KUKA KRL program: MyProgram_010().src

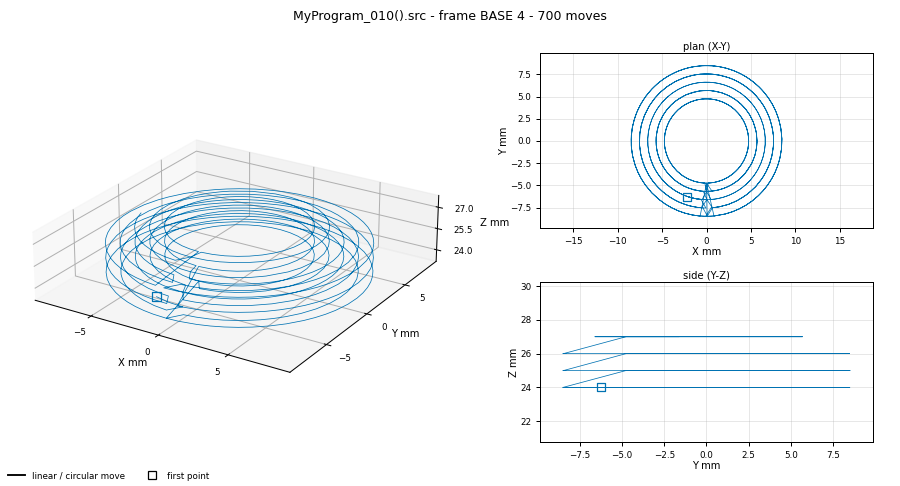
[picture p0: tool path of MyProgram_010().src in frame BASE 4, 700 of 700 moves have a stored position in this frame; points joined in program order, loops and branches not executed]
&ACCESS RVP
&REL 1
&PARAM TEMPLATE = C:\KRC\Roboter\Template\vorgabe
&PARAM EDITMASK = *
DEF MyProgram_010()
; ---- Setting reference (Base) ----
$BASE = BASE_DATA[4]

; --------------------------
; ---- Setting tool (TCP) ----
$TOOL = TOOL_DATA[3]
; --------------------------

$VEL.CP = VEL_APROX_PRINT
Startdeposition()
$VEL.CP = VEL_PRINT
LIN {X -2.1509,Y -6.2604,Z 24,A -3.0859,B 0,C 0,E1 0.1598,E2 90.0714} C_DIS
LIN {X -1.1022,Y -6.531,Z 24,A -3.0589,B 0,C 0,E1 0.1598,E2 90.0714} C_DIS
LIN {X 0.0303,Y -6.6205,Z 24,A -3.0212,B 0,C 0,E1 0.1598,E2 90.0715} C_DIS
Enddeposition()
LIN {X 0.0303,Y -6.6205,Z 24,A -3.0212,B 0,C 0,E1 0.1598,E2 90.0715} C_DIS
Startdeposition()
$VEL.CP = VEL_PRINT
LIN {X -0.5711,Y -7.5301,Z 24,A -3.0815,B 0,C 0,E1 0.1598,E2 90.0709} C_DIS
LIN {X -1.5725,Y -7.3914,Z 24,A -3.1128,B 0,C 0,E1 0.1598,E2 90.0714} C_DIS
LIN {X -2.6511,Y -7.0725,Z 24,A -3.1389,B 0,C 0,E1 0.1598,E2 90.0714} C_DIS
LIN {X -3.396,Y -6.7456,Z 24,A -3.1523,B 0,C 0,E1 0.1598,E2 90.0714} C_DIS
LIN {X -4.1021,Y -6.3418,Z 24,A -3.1611,B 0,C 0,E1 0.1598,E2 90.0713} C_DIS
LIN {X -4.7604,Y -5.8639,Z 24,A -3.165,B 0,C 0,E1 0.1598,E2 90.0713} C_DIS
LIN {X -5.3635,Y -5.318,Z 24,A -3.164,B 0,C 0,E1 0.1598,E2 90.0712} C_DIS
LIN {X -5.9042,Y -4.7103,Z 24,A -3.1581,B 0,C 0,E1 0.1598,E2 90.0712} C_DIS
LIN {X -6.3764,Y -4.048,Z 24,A -3.1474,B 0,C 0,E1 0.1598,E2 90.0712} C_DIS
LIN {X -6.7752,Y -3.339,Z 24,A -3.1321,B 0,C 0,E1 0.1598,E2 90.0712} C_DIS
LIN {X -7.1999,Y -2.2947,Z 24,A -3.1033,B 0,C 0,E1 0.1598,E2 90.0709} C_DIS
LIN {X -7.4401,Y -1.3287,Z 24,A -3.0713,B 0,C 0,E1 0.1598,E2 90.0709} C_DIS
LIN {X -7.5468,Y -0.4046,Z 24,A -3.0364,B 0,C 0,E1 0.1598,E2 90.0711} C_DIS
LIN {X -7.5022,Y 0.9089,Z 24,A -2.9788,B 0,C 0,E1 0.1598,E2 90.0706} C_DIS
LIN {X -7.3211,Y 1.8726,Z 24,A -2.9319,B 0,C 0,E1 0.1598,E2 90.0711} C_DIS
LIN {X -6.9098,Y 3.0609,Z 24,A -2.8664,B 0,C 0,E1 0.1598,E2 90.0711} C_DIS
LIN {X -6.4301,Y 3.9691,Z 24,A -2.8107,B 0,C 0,E1 0.1598,E2 90.0714} C_DIS
LIN {X -5.7251,Y 4.9319,Z 24,A -2.7441,B 0,C 0,E1 0.1598,E2 90.0714} C_DIS
LIN {X -5.1328,Y 5.5464,Z 24,A -2.6965,B 0,C 0,E1 0.1598,E2 90.0717} C_DIS
LIN {X -4.2881,Y 6.2219,Z 24,A -2.6369,B 0,C 0,E1 0.1598,E2 90.0718} C_DIS
LIN {X -3.4726,Y 6.7132,Z 24,A -2.5862,B 0,C 0,E1 0.1598,E2 90.072} C_DIS
LIN {X -2.6704,Y 7.0647,Z 24,A -2.5418,B 0,C 0,E1 0.1598,E2 90.0721} C_DIS
LIN {X -1.6242,Y 7.3805,Z 24,A -2.4898,B 0,C 0,E1 0.1598,E2 90.0722} C_DIS
LIN {X -0.7055,Y 7.5252,Z 24,A -2.4498,B 0,C 0,E1 0.1598,E2 90.0722} C_DIS
LIN {X 0.503,Y 7.5401,Z 24,A -2.4046,B 0,C 0,E1 0.1598,E2 90.0724} C_DIS
LIN {X 1.3896,Y 7.4296,Z 24,A -2.3765,B 0,C 0,E1 0.1598,E2 90.0724} C_DIS
LIN {X 2.6317,Y 7.0805,Z 24,A -2.3454,B 0,C 0,E1 0.1598,E2 90.0724} C_DIS
LIN {X 3.395,Y 6.7468,Z 24,A -2.3314,B 0,C 0,E1 0.1598,E2 90.0724} C_DIS
LIN {X 4.1176,Y 6.3321,Z 24,A -2.3223,B 0,C 0,E1 0.1598,E2 90.0724} C_DIS
LIN {X 4.7897,Y 5.8397,Z 24,A -2.3183,B 0,C 0,E1 0.1598,E2 90.0724} C_DIS
LIN {X 5.6394,Y 5.032,Z 24,A -2.321,B 0,C 0,E1 0.1598,E2 90.0721} C_DIS
LIN {X 6.3129,Y 4.149,Z 24,A -2.3336,B 0,C 0,E1 0.1598,E2 90.0721} C_DIS
LIN {X 6.6648,Y 3.5575,Z 24,A -2.346,B 0,C 0,E1 0.1598,E2 90.0722} C_DIS
LIN {X 7.0965,Y 2.5964,Z 24,A -2.3706,B 0,C 0,E1 0.1598,E2 90.0719} C_DIS
LIN {X 7.4222,Y 1.4016,Z 24,A -2.4091,B 0,C 0,E1 0.1598,E2 90.0715} C_DIS
LIN {X 7.5337,Y 0.5498,Z 24,A -2.4417,B 0,C 0,E1 0.1598,E2 90.0719} C_DIS
LIN {X 7.5455,Y -0.3091,Z 24,A -2.4778,B 0,C 0,E1 0.1598,E2 90.0719} C_DIS
LIN {X 7.4322,Y -1.3766,Z 24,A -2.5271,B 0,C 0,E1 0.1598,E2 90.0715} C_DIS
LIN {X 7.1168,Y -2.5308,Z 24,A -2.5877,B 0,C 0,E1 0.1598,E2 90.0713} C_DIS
LIN {X 6.6477,Y -3.5933,Z 24,A -2.6504,B 0,C 0,E1 0.1598,E2 90.0715} C_DIS
LIN {X 6.1054,Y -4.445,Z 24,A -2.7067,B 0,C 0,E1 0.1598,E2 90.0716} C_DIS
LIN {X 5.5965,Y -5.0722,Z 24,A -2.7522,B 0,C 0,E1 0.1598,E2 90.0716} C_DIS
LIN {X 5.0229,Y -5.641,Z 24,A -2.7975,B 0,C 0,E1 0.1598,E2 90.0716} C_DIS
LIN {X 4.1409,Y -6.3233,Z 24,A -2.8589,B 0,C 0,E1 0.1598,E2 90.0716} C_DIS
LIN {X 3.1206,Y -6.8785,Z 24,A -2.92,B 0,C 0,E1 0.1598,E2 90.0716} C_DIS
LIN {X 2.3301,Y -7.1857,Z 24,A -2.9621,B 0,C 0,E1 0.1598,E2 90.0716} C_DIS
LIN {X 1.5095,Y -7.3999,Z 24,A -3.0013,B 0,C 0,E1 0.1598,E2 90.0716} C_DIS
LIN {X 0.6704,Y -7.5218,Z 24,A -3.0373,B 0,C 0,E1 0.1598,E2 90.0716} C_DIS
LIN {X 0.6704,Y -7.5218,Z 24,A -3.0373,B 0,C 0,E1 0.1598,E2 90.0716} C_DIS
Enddeposition()
LIN {X 0.0638,Y -8.4902,Z 24,A -3.0997,B 0,C 0,E1 0.1598,E2 90.0703} C_DIS
Startdeposition()
$VEL.CP = VEL_PRINT
LIN {X 0.9236,Y -8.4401,Z 24,A -3.0671,B 0,C 0,E1 0.1598,E2 90.0714} C_DIS
LIN {X 2.0955,Y -8.2263,Z 24,A -3.0151,B 0,C 0,E1 0.1598,E2 90.0715} C_DIS
LIN {X 2.906,Y -7.9764,Z 24,A -2.9748,B 0,C 0,E1 0.1598,E2 90.0715} C_DIS
LIN {X 3.6874,Y -7.6466,Z 24,A -2.9321,B 0,C 0,E1 0.1598,E2 90.0716} C_DIS
LIN {X 4.432,Y -7.2405,Z 24,A -2.8875,B 0,C 0,E1 0.1598,E2 90.0716} C_DIS
LIN {X 5.1322,Y -6.7618,Z 24,A -2.8414,B 0,C 0,E1 0.1598,E2 90.0716} C_DIS
LIN {X 5.9363,Y -6.0709,Z 24,A -2.7823,B 0,C 0,E1 0.1598,E2 90.0716} C_DIS
LIN {X 6.6411,Y -5.2912,Z 24,A -2.7233,B 0,C 0,E1 0.1598,E2 90.0716} C_DIS
LIN {X 7.2908,Y -4.3455,Z 24,A -2.659,B 0,C 0,E1 0.1598,E2 90.0716} C_DIS
LIN {X 7.6767,Y -3.6219,Z 24,A -2.6142,B 0,C 0,E1 0.1598,E2 90.0718} C_DIS
LIN {X 7.9908,Y -2.8643,Z 24,A -2.5703,B 0,C 0,E1 0.1598,E2 90.0718} C_DIS
LIN {X 8.2302,Y -2.0798,Z 24,A -2.5281,B 0,C 0,E1 0.1598,E2 90.0718} C_DIS
LIN {X 8.4401,Y -0.9236,Z 24,A -2.4708,B 0,C 0,E1 0.1598,E2 90.0716} C_DIS
LIN {X 8.4863,Y 0.148,Z 24,A -2.4236,B 0,C 0,E1 0.1598,E2 90.0717} C_DIS
LIN {X 8.4278,Y 1.004,Z 24,A -2.3894,B 0,C 0,E1 0.1598,E2 90.072} C_DIS
LIN {X 8.2824,Y 1.8497,Z 24,A -2.3588,B 0,C 0,E1 0.1598,E2 90.072} C_DIS
LIN {X 8.0532,Y 2.6767,Z 24,A -2.3321,B 0,C 0,E1 0.1598,E2 90.072} C_DIS
LIN {X 7.7419,Y 3.4763,Z 24,A -2.3096,B 0,C 0,E1 0.1598,E2 90.0721} C_DIS
LIN {X 7.3514,Y 4.2404,Z 24,A -2.2915,B 0,C 0,E1 0.1598,E2 90.0721} C_DIS
LIN {X 6.8858,Y 4.9613,Z 24,A -2.2781,B 0,C 0,E1 0.1598,E2 90.0722} C_DIS
LIN {X 6.2076,Y 5.7923,Z 24,A -2.2676,B 0,C 0,E1 0.1598,E2 90.0721} C_DIS
LIN {X 5.4453,Y 6.5144,Z 24,A -2.2652,B 0,C 0,E1 0.1598,E2 90.0722} C_DIS
LIN {X 4.4548,Y 7.2234,Z 24,A -2.2717,B 0,C 0,E1 0.1598,E2 90.0722} C_DIS
LIN {X 3.733,Y 7.6202,Z 24,A -2.2817,B 0,C 0,E1 0.1598,E2 90.0724} C_DIS
LIN {X 2.9768,Y 7.9466,Z 24,A -2.2959,B 0,C 0,E1 0.1598,E2 90.0724} C_DIS
LIN {X 2.1925,Y 8.1983,Z 24,A -2.3142,B 0,C 0,E1 0.1598,E2 90.0724} C_DIS
LIN {X 1.3875,Y 8.3731,Z 24,A -2.3366,B 0,C 0,E1 0.1598,E2 90.0724} C_DIS
LIN {X 0.5694,Y 8.4695,Z 24,A -2.3627,B 0,C 0,E1 0.1598,E2 90.0724} C_DIS
LIN {X -0.4602,Y 8.4788,Z 24,A -2.4003,B 0,C 0,E1 0.1598,E2 90.0724} C_DIS
LIN {X -1.7187,Y 8.3132,Z 24,A -2.4538,B 0,C 0,E1 0.1598,E2 90.0723} C_DIS
LIN {X -2.5445,Y 8.0987,Z 24,A -2.4933,B 0,C 0,E1 0.1598,E2 90.0723} C_DIS
LIN {X -3.3445,Y 7.8021,Z 24,A -2.5354,B 0,C 0,E1 0.1598,E2 90.0722} C_DIS
LIN {X -4.1107,Y 7.4269,Z 24,A -2.5795,B 0,C 0,E1 0.1598,E2 90.0721} C_DIS
LIN {X -4.8354,Y 6.9766,Z 24,A -2.6252,B 0,C 0,E1 0.1598,E2 90.072} C_DIS
LIN {X -5.5111,Y 6.4557,Z 24,A -2.672,B 0,C 0,E1 0.1598,E2 90.0719} C_DIS
LIN {X -6.1312,Y 5.8697,Z 24,A -2.7196,B 0,C 0,E1 0.1598,E2 90.0718} C_DIS
LIN {X -6.8215,Y 5.0568,Z 24,A -2.7791,B 0,C 0,E1 0.1598,E2 90.0715} C_DIS
LIN {X -7.3978,Y 4.1667,Z 24,A -2.8378,B 0,C 0,E1 0.1598,E2 90.0714} C_DIS
LIN {X -7.8737,Y 3.1665,Z 24,A -2.8975,B 0,C 0,E1 0.1598,E2 90.0713} C_DIS
LIN {X -8.1612,Y 2.3284,Z 24,A -2.9435,B 0,C 0,E1 0.1598,E2 90.0713} C_DIS
LIN {X -8.3602,Y 1.4649,Z 24,A -2.9872,B 0,C 0,E1 0.1598,E2 90.0713} C_DIS
LIN {X -8.4687,Y 0.5855,Z 24,A -3.0282,B 0,C 0,E1 0.1598,E2 90.0711} C_DIS
LIN {X -8.4746,Y -0.5221,Z 24,A -3.0748,B 0,C 0,E1 0.1598,E2 90.0707} C_DIS
LIN {X -8.343,Y -1.5835,Z 24,A -3.1148,B 0,C 0,E1 0.1598,E2 90.0708} C_DIS
LIN {X -8.0507,Y -2.6866,Z 24,A -3.1506,B 0,C 0,E1 0.1598,E2 90.0707} C_DIS
LIN {X -7.7407,Y -3.4806,Z 24,A -3.173,B 0,C 0,E1 0.1598,E2 90.071} C_DIS
LIN {X -7.3527,Y -4.2396,Z 24,A -3.1909,B 0,C 0,E1 0.1598,E2 90.071} C_DIS
LIN {X -6.8904,Y -4.9557,Z 24,A -3.2042,B 0,C 0,E1 0.1598,E2 90.071} C_DIS
LIN {X -6.2176,Y -5.7818,Z 24,A -3.2143,B 0,C 0,E1 0.1598,E2 90.0709} C_DIS
LIN {X -5.4465,Y -6.5135,Z 24,A -3.217,B 0,C 0,E1 0.1598,E2 90.0709} C_DIS
LIN {X -4.6444,Y -7.103,Z 24,A -3.2127,B 0,C 0,E1 0.1598,E2 90.0711} C_DIS
LIN {X -3.9579,Y -7.5063,Z 24,A -3.2047,B 0,C 0,E1 0.1598,E2 90.0712} C_DIS
LIN {X -3.2368,Y -7.8438,Z 24,A -3.1926,B 0,C 0,E1 0.1598,E2 90.0712} C_DIS
LIN {X -2.4874,Y -8.1126,Z 24,A -3.1765,B 0,C 0,E1 0.1598,E2 90.0712} C_DIS
LIN {X -1.7162,Y -8.3104,Z 24,A -3.1567,B 0,C 0,E1 0.1598,E2 90.0713} C_DIS
LIN {X -0.9299,Y -8.4356,Z 24,A -3.1332,B 0,C 0,E1 0.1598,E2 90.0713} C_DIS
LIN {X 0.0638,Y -8.4902,Z 24,A -3.0991,B 0,C 0,E1 0.1598,E2 90.0714} C_DIS
Enddeposition()
LIN {X 0.0007,Y -4.7572,Z 25,A -2.9279,B 0,C 0,E1 0.1598,E2 90.0604} C_DIS
Startdeposition()
$VEL.CP = VEL_PRINT
LIN {X 0.0007,Y -4.7572,Z 25,A -2.9336,B 0,C 0,E1 0.1598,E2 90.0661} C_DIS
LIN {X -0.6666,Y -4.7028,Z 25,A -2.9607,B 0,C 0,E1 0.1598,E2 90.071} C_DIS
LIN {X -1.3207,Y -4.5622,Z 25,A -2.9794,B 0,C 0,E1 0.1598,E2 90.0715} C_DIS
LIN {X -2.0351,Y -4.2906,Z 25,A -2.9941,B 0,C 0,E1 0.1598,E2 90.0715} C_DIS
LIN {X -2.6974,Y -3.909,Z 25,A -3.0022,B 0,C 0,E1 0.1598,E2 90.0715} C_DIS
LIN {X -3.2894,Y -3.4255,Z 25,A -3.0034,B 0,C 0,E1 0.1598,E2 90.0715} C_DIS
LIN {X -3.679,Y -3.0044,Z 25,A -3,B 0,C 0,E1 0.1598,E2 90.0715} C_DIS
LIN {X -4.112,Y -2.3746,Z 25,A -2.9891,B 0,C 0,E1 0.1598,E2 90.0714} C_DIS
LIN {X -4.3699,Y -1.8625,Z 25,A -2.9769,B 0,C 0,E1 0.1598,E2 90.0714} C_DIS
LIN {X -4.6107,Y -1.137,Z 25,A -2.955,B 0,C 0,E1 0.1598,E2 90.0714} C_DIS
LIN {X -4.7143,Y -0.5729,Z 25,A -2.935,B 0,C 0,E1 0.1598,E2 90.0714} C_DIS
LIN {X -4.75,Y -0.0006,Z 25,A -2.9122,B 0,C 0,E1 0.1598,E2 90.0715} C_DIS
LIN {X -4.69,Y 0.7615,Z 25,A -2.8777,B 0,C 0,E1 0.1598,E2 90.0715} C_DIS
LIN {X -4.5075,Y 1.5041,Z 25,A -2.8396,B 0,C 0,E1 0.1598,E2 90.0715} C_DIS
LIN {X -4.2076,Y 2.2075,Z 25,A -2.7988,B 0,C 0,E1 0.1598,E2 90.0715} C_DIS
LIN {X -3.7991,Y 2.8541,Z 25,A -2.7565,B 0,C 0,E1 0.1598,E2 90.0717} C_DIS
LIN {X -3.221,Y 3.4906,Z 25,A -2.7083,B 0,C 0,E1 0.1598,E2 90.0717} C_DIS
LIN {X -2.6984,Y 3.9084,Z 25,A -2.6715,B 0,C 0,E1 0.1598,E2 90.0719} C_DIS
LIN {X -2.0366,Y 4.2911,Z 25,A -2.631,B 0,C 0,E1 0.1598,E2 90.0719} C_DIS
LIN {X -1.3226,Y 4.5641,Z 25,A -2.5931,B 0,C 0,E1 0.1598,E2 90.0721} C_DIS
LIN {X -0.5734,Y 4.7175,Z 25,A -2.559,B 0,C 0,E1 0.1598,E2 90.0721} C_DIS
LIN {X 0.1908,Y 4.7483,Z 25,A -2.5296,B 0,C 0,E1 0.1598,E2 90.0721} C_DIS
LIN {X 0.9495,Y 4.6541,Z 25,A -2.5056,B 0,C 0,E1 0.1598,E2 90.0722} C_DIS
LIN {X 1.6835,Y 4.4406,Z 25,A -2.4876,B 0,C 0,E1 0.1598,E2 90.0722} C_DIS
LIN {X 2.3736,Y 4.1125,Z 25,A -2.476,B 0,C 0,E1 0.1598,E2 90.0722} C_DIS
LIN {X 3.0036,Y 3.6797,Z 25,A -2.4711,B 0,C 0,E1 0.1598,E2 90.0722} C_DIS
LIN {X 3.5539,Y 3.1492,Z 25,A -2.4732,B 0,C 0,E1 0.1598,E2 90.0722} C_DIS
LIN {X 4.014,Y 2.5391,Z 25,A -2.4821,B 0,C 0,E1 0.1598,E2 90.072} C_DIS
LIN {X 4.3693,Y 1.8622,Z 25,A -2.4977,B 0,C 0,E1 0.1598,E2 90.072} C_DIS
LIN {X 4.6107,Y 1.137,Z 25,A -2.5196,B 0,C 0,E1 0.1598,E2 90.072} C_DIS
LIN {X 4.7339,Y 0.3828,Z 25,A -2.5471,B 0,C 0,E1 0.1598,E2 90.0719} C_DIS
LIN {X 4.7339,Y -0.3814,Z 25,A -2.5795,B 0,C 0,E1 0.1598,E2 90.0719} C_DIS
LIN {X 4.654,Y -0.9495,Z 25,A -2.6068,B 0,C 0,E1 0.1598,E2 90.0719} C_DIS
LIN {X 4.4402,Y -1.6832,Z 25,A -2.6457,B 0,C 0,E1 0.1598,E2 90.0718} C_DIS
LIN {X 4.2062,Y -2.2067,Z 25,A -2.6767,B 0,C 0,E1 0.1598,E2 90.0718} C_DIS
LIN {X 3.7983,Y -2.8534,Z 25,A -2.7191,B 0,C 0,E1 0.1598,E2 90.0718} C_DIS
LIN {X 3.2912,Y -3.4257,Z 25,A -2.7621,B 0,C 0,E1 0.1598,E2 90.0718} C_DIS
LIN {X 2.6986,Y -3.9082,Z 25,A -2.8044,B 0,C 0,E1 0.1598,E2 90.0718} C_DIS
LIN {X 2.0365,Y -4.2902,Z 25,A -2.845,B 0,C 0,E1 0.1598,E2 90.0718} C_DIS
LIN {X 1.3221,Y -4.5618,Z 25,A -2.8828,B 0,C 0,E1 0.1598,E2 90.0717} C_DIS
LIN {X 0.5734,Y -4.7168,Z 25,A -2.9168,B 0,C 0,E1 0.1598,E2 90.0717} C_DIS
LIN {X 0.0007,Y -4.7572,Z 25,A -2.9396,B 0,C 0,E1 0.1598,E2 90.0717} C_DIS
Enddeposition()
LIN {X 0.0007,Y -4.7572,Z 25,A -2.9396,B 0,C 0,E1 0.1598,E2 90.0717} C_DIS
Startdeposition()
$VEL.CP = VEL_PRINT
LIN {X 0.6179,Y -5.6511,Z 25,A -2.9544,B 0,C 0,E1 0.1598,E2 90.0711} C_DIS
LIN {X 1.4035,Y -5.5101,Z 25,A -2.9201,B 0,C 0,E1 0.1598,E2 90.0716} C_DIS
LIN {X 2.1613,Y -5.2591,Z 25,A -2.8817,B 0,C 0,E1 0.1598,E2 90.0717} C_DIS
LIN {X 2.8755,Y -4.9034,Z 25,A -2.8403,B 0,C 0,E1 0.1598,E2 90.0717} C_DIS
LIN {X 3.5341,Y -4.4526,Z 25,A -2.7969,B 0,C 0,E1 0.1598,E2 90.0717} C_DIS
LIN {X 4.2617,Y -3.7701,Z 25,A -2.741,B 0,C 0,E1 0.1598,E2 90.0717} C_DIS
LIN {X 5.0937,Y -2.5348,Z 25,A -2.6575,B 0,C 0,E1 0.1598,E2 90.0713} C_DIS
LIN {X 5.4673,Y -1.5791,Z 25,A -2.6033,B 0,C 0,E1 0.1598,E2 90.0716} C_DIS
LIN {X 5.6386,Y -0.7147,Z 25,A -2.5604,B 0,C 0,E1 0.1598,E2 90.0718} C_DIS
LIN {X 5.6861,Y -0.0114,Z 25,A -2.5289,B 0,C 0,E1 0.1598,E2 90.0719} C_DIS
LIN {X 5.5965,Y 1.0311,Z 25,A -2.4875,B 0,C 0,E1 0.1598,E2 90.0717} C_DIS
LIN {X 5.2553,Y 2.162,Z 25,A -2.4519,B 0,C 0,E1 0.1598,E2 90.0716} C_DIS
LIN {X 4.8879,Y 2.8991,Z 25,A -2.4345,B 0,C 0,E1 0.1598,E2 90.072} C_DIS
LIN {X 4.4167,Y 3.5747,Z 25,A -2.4232,B 0,C 0,E1 0.1598,E2 90.072} C_DIS
LIN {X 3.854,Y 4.1761,Z 25,A -2.4185,B 0,C 0,E1 0.1598,E2 90.0721} C_DIS
LIN {X 3.2096,Y 4.689,Z 25,A -2.4206,B 0,C 0,E1 0.1598,E2 90.0721} C_DIS
LIN {X 2.4982,Y 5.104,Z 25,A -2.4293,B 0,C 0,E1 0.1598,E2 90.0722} C_DIS
LIN {X 1.7342,Y 5.4121,Z 25,A -2.4444,B 0,C 0,E1 0.1598,E2 90.0722} C_DIS
LIN {X 0.9339,Y 5.6074,Z 25,A -2.4657,B 0,C 0,E1 0.1598,E2 90.0722} C_DIS
LIN {X 0.1135,Y 5.684,Z 25,A -2.4927,B 0,C 0,E1 0.1598,E2 90.0722} C_DIS
LIN {X -0.7093,Y 5.6404,Z 25,A -2.5249,B 0,C 0,E1 0.1598,E2 90.0722} C_DIS
LIN {X -1.5169,Y 5.4776,Z 25,A -2.5616,B 0,C 0,E1 0.1598,E2 90.0722} C_DIS
LIN {X -2.2929,Y 5.2012,Z 25,A -2.6019,B 0,C 0,E1 0.1598,E2 90.0721} C_DIS
LIN {X -3.0203,Y 4.8143,Z 25,A -2.645,B 0,C 0,E1 0.1598,E2 90.072} C_DIS
LIN {X -3.6839,Y 4.3264,Z 25,A -2.69,B 0,C 0,E1 0.1598,E2 90.0719} C_DIS
LIN {X -4.2727,Y 3.7502,Z 25,A -2.736,B 0,C 0,E1 0.1598,E2 90.0718} C_DIS
LIN {X -4.7695,Y 3.093,Z 25,A -2.782,B 0,C 0,E1 0.1598,E2 90.0716} C_DIS
LIN {X -5.1668,Y 2.3713,Z 25,A -2.8271,B 0,C 0,E1 0.1598,E2 90.0716} C_DIS
LIN {X -5.4558,Y 1.5998,Z 25,A -2.8703,B 0,C 0,E1 0.1598,E2 90.0714} C_DIS
LIN {X -5.6305,Y 0.7944,Z 25,A -2.9107,B 0,C 0,E1 0.1598,E2 90.0714} C_DIS
LIN {X -5.6864,Y -0.0279,Z 25,A -2.9474,B 0,C 0,E1 0.1598,E2 90.0713} C_DIS
LIN {X -5.62,Y -0.8492,Z 25,A -2.9797,B 0,C 0,E1 0.1598,E2 90.0713} C_DIS
LIN {X -5.4383,Y -1.6526,Z 25,A -3.007,B 0,C 0,E1 0.1598,E2 90.0713} C_DIS
LIN {X -5.1415,Y -2.421,Z 25,A -3.0286,B 0,C 0,E1 0.1598,E2 90.0713} C_DIS
LIN {X -4.7374,Y -3.1388,Z 25,A -3.0441,B 0,C 0,E1 0.1598,E2 90.0713} C_DIS
LIN {X -4.2335,Y -3.7903,Z 25,A -3.0532,B 0,C 0,E1 0.1598,E2 90.0713} C_DIS
LIN {X -3.6412,Y -4.3627,Z 25,A -3.0557,B 0,C 0,E1 0.1598,E2 90.0713} C_DIS
LIN {X -2.9718,Y -4.8422,Z 25,A -3.0515,B 0,C 0,E1 0.1598,E2 90.0713} C_DIS
LIN {X -2.242,Y -5.2243,Z 25,A -3.0409,B 0,C 0,E1 0.1598,E2 90.0714} C_DIS
LIN {X -1.4324,Y -5.5062,Z 25,A -3.0232,B 0,C 0,E1 0.1598,E2 90.0714} C_DIS
LIN {X -0.3615,Y -5.6758,Z 25,A -2.9911,B 0,C 0,E1 0.1598,E2 90.0716} C_DIS
LIN {X -0.3615,Y -5.6758,Z 25,A -2.9911,B 0,C 0,E1 0.1598,E2 90.0716} C_DIS
Enddeposition()
LIN {X 0.0548,Y -6.6232,Z 25,A -3.0151,B 0,C 0,E1 0.1598,E2 90.0704} C_DIS
Startdeposition()
$VEL.CP = VEL_PRINT
LIN {X -0.8791,Y -6.559,Z 25,A -3.0477,B 0,C 0,E1 0.1598,E2 90.0714} C_DIS
LIN {X -1.6146,Y -6.4178,Z 25,A -3.0687,B 0,C 0,E1 0.1598,E2 90.0714} C_DIS
LIN {X -2.3305,Y -6.1976,Z 25,A -3.0857,B 0,C 0,E1 0.1598,E2 90.0714} C_DIS
LIN {X -3.0152,Y -5.8938,Z 25,A -3.0979,B 0,C 0,E1 0.1598,E2 90.0714} C_DIS
LIN {X -3.6616,Y -5.5156,Z 25,A -3.1056,B 0,C 0,E1 0.1598,E2 90.0714} C_DIS
LIN {X -4.2617,Y -5.0673,Z 25,A -3.1086,B 0,C 0,E1 0.1598,E2 90.0714} C_DIS
LIN {X -4.8059,Y -4.5527,Z 25,A -3.1067,B 0,C 0,E1 0.1598,E2 90.0713} C_DIS
LIN {X -5.2881,Y -3.9794,Z 25,A -3.1002,B 0,C 0,E1 0.1598,E2 90.0713} C_DIS
LIN {X -5.7046,Y -3.3569,Z 25,A -3.0891,B 0,C 0,E1 0.1598,E2 90.0713} C_DIS
LIN {X -6.0462,Y -2.6904,Z 25,A -3.0734,B 0,C 0,E1 0.1598,E2 90.0713} C_DIS
LIN {X -6.3118,Y -1.9902,Z 25,A -3.0536,B 0,C 0,E1 0.1598,E2 90.0713} C_DIS
LIN {X -6.4964,Y -1.2643,Z 25,A -3.0297,B 0,C 0,E1 0.1598,E2 90.0713} C_DIS
LIN {X -6.5973,Y -0.5223,Z 25,A -3.0021,B 0,C 0,E1 0.1598,E2 90.0713} C_DIS
LIN {X -6.6169,Y 0.2265,Z 25,A -2.9712,B 0,C 0,E1 0.1598,E2 90.0713} C_DIS
LIN {X -6.5466,Y 0.9722,Z 25,A -2.9371,B 0,C 0,E1 0.1598,E2 90.0713} C_DIS
LIN {X -6.394,Y 1.7054,Z 25,A -2.9005,B 0,C 0,E1 0.1598,E2 90.0714} C_DIS
LIN {X -6.1631,Y 2.4178,Z 25,A -2.862,B 0,C 0,E1 0.1598,E2 90.0714} C_DIS
LIN {X -5.8507,Y 3.0986,Z 25,A -2.8218,B 0,C 0,E1 0.1598,E2 90.0716} C_DIS
LIN {X -5.4642,Y 3.7402,Z 25,A -2.7805,B 0,C 0,E1 0.1598,E2 90.0716} C_DIS
LIN {X -5.0067,Y 4.3333,Z 25,A -2.7386,B 0,C 0,E1 0.1598,E2 90.0717} C_DIS
LIN {X -4.4845,Y 4.8704,Z 25,A -2.6967,B 0,C 0,E1 0.1598,E2 90.0718} C_DIS
LIN {X -3.9053,Y 5.3451,Z 25,A -2.6553,B 0,C 0,E1 0.1598,E2 90.0719} C_DIS
LIN {X -3.2761,Y 5.7514,Z 25,A -2.615,B 0,C 0,E1 0.1598,E2 90.072} C_DIS
LIN {X -2.6047,Y 6.0832,Z 25,A -2.5762,B 0,C 0,E1 0.1598,E2 90.072} C_DIS
LIN {X -1.9013,Y 6.3404,Z 25,A -2.5394,B 0,C 0,E1 0.1598,E2 90.0722} C_DIS
LIN {X -1.1732,Y 6.5159,Z 25,A -2.5052,B 0,C 0,E1 0.1598,E2 90.0722} C_DIS
LIN {X -0.4294,Y 6.6037,Z 25,A -2.474,B 0,C 0,E1 0.1598,E2 90.0722} C_DIS
LIN {X 0.3194,Y 6.6111,Z 25,A -2.4461,B 0,C 0,E1 0.1598,E2 90.0723} C_DIS
LIN {X 1.0644,Y 6.5338,Z 25,A -2.4219,B 0,C 0,E1 0.1598,E2 90.0723} C_DIS
LIN {X 1.7954,Y 6.3703,Z 25,A -2.4018,B 0,C 0,E1 0.1598,E2 90.0723} C_DIS
LIN {X 2.5037,Y 6.1273,Z 25,A -2.386,B 0,C 0,E1 0.1598,E2 90.0723} C_DIS
LIN {X 3.1793,Y 5.804,Z 25,A -2.3747,B 0,C 0,E1 0.1598,E2 90.0723} C_DIS
LIN {X 3.8145,Y 5.4074,Z 25,A -2.3681,B 0,C 0,E1 0.1598,E2 90.0723} C_DIS
LIN {X 4.4022,Y 4.9431,Z 25,A -2.3661,B 0,C 0,E1 0.1598,E2 90.0723} C_DIS
LIN {X 4.9326,Y 4.4142,Z 25,A -2.3689,B 0,C 0,E1 0.1598,E2 90.0723} C_DIS
LIN {X 5.399,Y 3.828,Z 25,A -2.3766,B 0,C 0,E1 0.1598,E2 90.0722} C_DIS
LIN {X 5.7968,Y 3.1934,Z 25,A -2.3888,B 0,C 0,E1 0.1598,E2 90.0722} C_DIS
LIN {X 6.1208,Y 2.5182,Z 25,A -2.4056,B 0,C 0,E1 0.1598,E2 90.0721} C_DIS
LIN {X 6.3667,Y 1.8107,Z 25,A -2.4265,B 0,C 0,E1 0.1598,E2 90.0721} C_DIS
LIN {X 6.533,Y 1.0803,Z 25,A -2.4515,B 0,C 0,E1 0.1598,E2 90.072} C_DIS
LIN {X 6.6101,Y 0.3352,Z 25,A -2.4803,B 0,C 0,E1 0.1598,E2 90.072} C_DIS
LIN {X 6.6063,Y -0.4136,Z 25,A -2.5123,B 0,C 0,E1 0.1598,E2 90.072} C_DIS
LIN {X 6.5152,Y -1.157,Z 25,A -2.5472,B 0,C 0,E1 0.1598,E2 90.0719} C_DIS
LIN {X 6.3441,Y -1.8862,Z 25,A -2.5846,B 0,C 0,E1 0.1598,E2 90.0719} C_DIS
LIN {X 6.0916,Y -2.5914,Z 25,A -2.6239,B 0,C 0,E1 0.1598,E2 90.0719} C_DIS
LIN {X 5.7607,Y -3.2633,Z 25,A -2.6646,B 0,C 0,E1 0.1598,E2 90.0718} C_DIS
LIN {X 5.354,Y -3.8922,Z 25,A -2.7064,B 0,C 0,E1 0.1598,E2 90.0718} C_DIS
LIN {X 4.8809,Y -4.4728,Z 25,A -2.7485,B 0,C 0,E1 0.1598,E2 90.0718} C_DIS
LIN {X 4.3449,Y -4.9961,Z 25,A -2.7904,B 0,C 0,E1 0.1598,E2 90.0718} C_DIS
LIN {X 3.7533,Y -5.4556,Z 25,A -2.8317,B 0,C 0,E1 0.1598,E2 90.0717} C_DIS
LIN {X 3.1125,Y -5.8435,Z 25,A -2.8717,B 0,C 0,E1 0.1598,E2 90.0717} C_DIS
LIN {X 2.4324,Y -6.1573,Z 25,A -2.9101,B 0,C 0,E1 0.1598,E2 90.0717} C_DIS
LIN {X 1.7206,Y -6.3902,Z 25,A -2.9461,B 0,C 0,E1 0.1598,E2 90.0717} C_DIS
LIN {X 0.9877,Y -6.5443,Z 25,A -2.9795,B 0,C 0,E1 0.1598,E2 90.0716} C_DIS
LIN {X 0.0548,Y -6.6232,Z 25,A -3.0171,B 0,C 0,E1 0.1598,E2 90.0716} C_DIS
Enddeposition()
LIN {X 0.0548,Y -6.6232,Z 25,A -3.0171,B 0,C 0,E1 0.1598,E2 90.0716} C_DIS
Startdeposition()
$VEL.CP = VEL_PRINT
LIN {X 0.6647,Y -7.5237,Z 25,A -3.0326,B 0,C 0,E1 0.1598,E2 90.071} C_DIS
LIN {X 1.4283,Y -7.4179,Z 25,A -3.0006,B 0,C 0,E1 0.1598,E2 90.0715} C_DIS
LIN {X 2.487,Y -7.1368,Z 25,A -2.9499,B 0,C 0,E1 0.1598,E2 90.0716} C_DIS
LIN {X 3.476,Y -6.7112,Z 25,A -2.8954,B 0,C 0,E1 0.1598,E2 90.0716} C_DIS
LIN {X 4.5755,Y -6.0138,Z 25,A -2.8253,B 0,C 0,E1 0.1598,E2 90.0716} C_DIS
LIN {X 5.5309,Y -5.1492,Z 25,A -2.7533,B 0,C 0,E1 0.1598,E2 90.0716} C_DIS
LIN {X 6.3031,Y -4.1622,Z 25,A -2.6828,B 0,C 0,E1 0.1598,E2 90.0715} C_DIS
LIN {X 6.7424,Y -3.4026,Z 25,A -2.6345,B 0,C 0,E1 0.1598,E2 90.0717} C_DIS
LIN {X 7.0936,Y -2.5985,Z 25,A -2.5873,B 0,C 0,E1 0.1598,E2 90.0717} C_DIS
LIN {X 7.3457,Y -1.758,Z 25,A -2.5423,B 0,C 0,E1 0.1598,E2 90.0717} C_DIS
LIN {X 7.5347,Y -0.5845,Z 25,A -2.485,B 0,C 0,E1 0.1598,E2 90.0716} C_DIS
LIN {X 7.533,Y 0.536,Z 25,A -2.4374,B 0,C 0,E1 0.1598,E2 90.0716} C_DIS
LIN {X 7.4317,Y 1.3396,Z 25,A -2.4073,B 0,C 0,E1 0.1598,E2 90.072} C_DIS
LIN {X 7.0851,Y 2.6275,Z 25,A -2.3647,B 0,C 0,E1 0.1598,E2 90.0714} C_DIS
LIN {X 6.5609,Y 3.7512,Z 25,A -2.3364,B 0,C 0,E1 0.1598,E2 90.0717} C_DIS
LIN {X 5.9672,Y 4.6299,Z 25,A -2.3212,B 0,C 0,E1 0.1598,E2 90.072} C_DIS
LIN {X 5.2461,Y 5.4389,Z 25,A -2.3136,B 0,C 0,E1 0.1598,E2 90.072} C_DIS
LIN {X 4.5595,Y 6.0262,Z 25,A -2.3142,B 0,C 0,E1 0.1598,E2 90.0723} C_DIS
LIN {X 3.634,Y 6.6219,Z 25,A -2.323,B 0,C 0,E1 0.1598,E2 90.0723} C_DIS
LIN {X 2.9408,Y 6.9599,Z 25,A -2.3344,B 0,C 0,E1 0.1598,E2 90.0723} C_DIS
LIN {X 2.0312,Y 7.2798,Z 25,A -2.3544,B 0,C 0,E1 0.1598,E2 90.0723} C_DIS
LIN {X 0.6647,Y 7.5292,Z 25,A -2.3943,B 0,C 0,E1 0.1598,E2 90.0723} C_DIS
LIN {X -0.7155,Y 7.524,Z 25,A -2.4456,B 0,C 0,E1 0.1598,E2 90.0723} C_DIS
LIN {X -1.7089,Y 7.3627,Z 25,A -2.489,B 0,C 0,E1 0.1598,E2 90.0723} C_DIS
LIN {X -2.6446,Y 7.073,Z 25,A -2.5358,B 0,C 0,E1 0.1598,E2 90.0722} C_DIS
LIN {X -3.5402,Y 6.6768,Z 25,A -2.5855,B 0,C 0,E1 0.1598,E2 90.072} C_DIS
LIN {X -4.4964,Y 6.0747,Z 25,A -2.6461,B 0,C 0,E1 0.1598,E2 90.0719} C_DIS
LIN {X -5.21,Y 5.4731,Z 25,A -2.6978,B 0,C 0,E1 0.1598,E2 90.0718} C_DIS
LIN {X -5.8734,Y 4.7577,Z 25,A -2.7524,B 0,C 0,E1 0.1598,E2 90.0717} C_DIS
LIN {X -6.4706,Y 3.9036,Z 25,A -2.8103,B 0,C 0,E1 0.1598,E2 90.0715} C_DIS
LIN {X -7.0079,Y 2.8188,Z 25,A -2.8756,B 0,C 0,E1 0.1598,E2 90.0711} C_DIS
LIN {X -7.3607,Y 1.718,Z 25,A -2.935,B 0,C 0,E1 0.1598,E2 90.0711} C_DIS
LIN {X -7.5287,Y 0.6717,Z 25,A -2.9854,B 0,C 0,E1 0.1598,E2 90.0711} C_DIS
LIN {X -7.5415,Y -0.483,Z 25,A -3.0345,B 0,C 0,E1 0.1598,E2 90.0709} C_DIS
LIN {X -7.373,Y -1.6413,Z 25,A -3.0772,B 0,C 0,E1 0.1598,E2 90.0709} C_DIS
LIN {X -7.0154,Y -2.8124,Z 25,A -3.1135,B 0,C 0,E1 0.1598,E2 90.0708} C_DIS
LIN {X -6.5706,Y -3.7271,Z 25,A -3.136,B 0,C 0,E1 0.1598,E2 90.071} C_DIS
LIN {X -6.1308,Y -4.4118,Z 25,A -3.149,B 0,C 0,E1 0.1598,E2 90.0711} C_DIS
LIN {X -5.6205,Y -5.0456,Z 25,A -3.1571,B 0,C 0,E1 0.1598,E2 90.0711} C_DIS
LIN {X -5.0445,Y -5.6202,Z 25,A -3.1603,B 0,C 0,E1 0.1598,E2 90.0711} C_DIS
LIN {X -4.4106,Y -6.1302,Z 25,A -3.1586,B 0,C 0,E1 0.1598,E2 90.0712} C_DIS
LIN {X -3.7255,Y -6.569,Z 25,A -3.1521,B 0,C 0,E1 0.1598,E2 90.0712} C_DIS
LIN {X -2.997,Y -6.9312,Z 25,A -3.1408,B 0,C 0,E1 0.1598,E2 90.0713} C_DIS
LIN {X -2.0408,Y -7.2773,Z 25,A -3.1204,B 0,C 0,E1 0.1598,E2 90.0713} C_DIS
LIN {X -1.048,Y -7.4809,Z 25,A -3.0927,B 0,C 0,E1 0.1598,E2 90.0714} C_DIS
LIN {X -0.4005,Y -7.5423,Z 25,A -3.0716,B 0,C 0,E1 0.1598,E2 90.0714} C_DIS
LIN {X -0.4005,Y -7.5423,Z 25,A -3.0716,B 0,C 0,E1 0.1598,E2 90.0714} C_DIS
Enddeposition()
LIN {X 0.1112,Y -8.4893,Z 25,A -3.092,B 0,C 0,E1 0.1598,E2 90.0703} C_DIS
Startdeposition()
$VEL.CP = VEL_PRINT
LIN {X -0.8947,Y -8.4391,Z 25,A -3.1279,B 0,C 0,E1 0.1598,E2 90.0713} C_DIS
LIN {X -1.6909,Y -8.3155,Z 25,A -3.1519,B 0,C 0,E1 0.1598,E2 90.0713} C_DIS
LIN {X -2.4718,Y -8.1174,Z 25,A -3.1721,B 0,C 0,E1 0.1598,E2 90.0713} C_DIS
LIN {X -3.2306,Y -7.8464,Z 25,A -3.1884,B 0,C 0,E1 0.1598,E2 90.0713} C_DIS
LIN {X -3.9604,Y -7.5049,Z 25,A -3.2006,B 0,C 0,E1 0.1598,E2 90.0713} C_DIS
LIN {X -4.6547,Y -7.0959,Z 25,A -3.2087,B 0,C 0,E1 0.1598,E2 90.0713} C_DIS
LIN {X -5.3074,Y -6.6232,Z 25,A -3.2126,B 0,C 0,E1 0.1598,E2 90.0712} C_DIS
LIN {X -6.1421,Y -5.8613,Z 25,A -3.2108,B 0,C 0,E1 0.1598,E2 90.071} C_DIS
LIN {X -6.885,Y -4.9631,Z 25,A -3.2,B 0,C 0,E1 0.1598,E2 90.0708} C_DIS
LIN {X -7.3467,Y -4.2498,Z 25,A -3.187,B 0,C 0,E1 0.1598,E2 90.071} C_DIS
LIN {X -7.7348,Y -3.4941,Z 25,A -3.1693,B 0,C 0,E1 0.1598,E2 90.071} C_DIS
LIN {X -8.0448,Y -2.7031,Z 25,A -3.1472,B 0,C 0,E1 0.1598,E2 90.071} C_DIS
LIN {X -8.3231,Y -1.6784,Z 25,A -3.1139,B 0,C 0,E1 0.1598,E2 90.0708} C_DIS
LIN {X -8.4621,Y -0.708,Z 25,A -3.0782,B 0,C 0,E1 0.1598,E2 90.071} C_DIS
LIN {X -8.4675,Y 0.6023,Z 25,A -3.0227,B 0,C 0,E1 0.1598,E2 90.0707} C_DIS
LIN {X -8.3568,Y 1.4826,Z 25,A -2.982,B 0,C 0,E1 0.1598,E2 90.0712} C_DIS
LIN {X -8.1554,Y 2.3466,Z 25,A -2.9382,B 0,C 0,E1 0.1598,E2 90.0712} C_DIS
LIN {X -7.8656,Y 3.1851,Z 25,A -2.8922,B 0,C 0,E1 0.1598,E2 90.0714} C_DIS
LIN {X -7.4902,Y 3.989,Z 25,A -2.8445,B 0,C 0,E1 0.1598,E2 90.0714} C_DIS
LIN {X -6.8358,Y 5.0382,Z 25,A -2.7759,B 0,C 0,E1 0.1598,E2 90.0714} C_DIS
LIN {X -6.146,Y 5.8536,Z 25,A -2.7163,B 0,C 0,E1 0.1598,E2 90.0716} C_DIS
LIN {X -5.5264,Y 6.4419,Z 25,A -2.6688,B 0,C 0,E1 0.1598,E2 90.0718} C_DIS
LIN {X -4.851,Y 6.9651,Z 25,A -2.6218,B 0,C 0,E1 0.1598,E2 90.0719} C_DIS
LIN {X -4.1263,Y 7.4177,Z 25,A -2.576,B 0,C 0,E1 0.1598,E2 90.072} C_DIS
LIN {X -3.0919,Y 7.9091,Z 25,A -2.5171,B 0,C 0,E1 0.1598,E2 90.0721} C_DIS
LIN {X -2.0997,Y 8.2254,Z 25,A -2.4672,B 0,C 0,E1 0.1598,E2 90.0722} C_DIS
LIN {X -1.2831,Y 8.3913,Z 25,A -2.43,B 0,C 0,E1 0.1598,E2 90.0723} C_DIS
LIN {X -0.0341,Y 8.4919,Z 25,A -2.3797,B 0,C 0,E1 0.1598,E2 90.0723} C_DIS
LIN {X 0.991,Y 8.4301,Z 25,A -2.3444,B 0,C 0,E1 0.1598,E2 90.0724} C_DIS
LIN {X 1.8012,Y 8.2936,Z 25,A -2.3203,B 0,C 0,E1 0.1598,E2 90.0724} C_DIS
LIN {X 2.5945,Y 8.0798,Z 25,A -2.3,B 0,C 0,E1 0.1598,E2 90.0724} C_DIS
LIN {X 3.3634,Y 7.7907,Z 25,A -2.2838,B 0,C 0,E1 0.1598,E2 90.0724} C_DIS
LIN {X 4.1008,Y 7.4286,Z 25,A -2.2719,B 0,C 0,E1 0.1598,E2 90.0724} C_DIS
LIN {X 4.9716,Y 6.8844,Z 25,A -2.2627,B 0,C 0,E1 0.1598,E2 90.0724} C_DIS
LIN {X 5.9193,Y 6.0835,Z 25,A -2.2616,B 0,C 0,E1 0.1598,E2 90.0721} C_DIS
LIN {X 6.4978,Y 5.462,Z 25,A -2.2668,B 0,C 0,E1 0.1598,E2 90.0723} C_DIS
LIN {X 7.0113,Y 4.7858,Z 25,A -2.2765,B 0,C 0,E1 0.1598,E2 90.0723} C_DIS
LIN {X 7.4544,Y 4.0616,Z 25,A -2.291,B 0,C 0,E1 0.1598,E2 90.0722} C_DIS
LIN {X 7.8229,Y 3.2967,Z 25,A -2.3099,B 0,C 0,E1 0.1598,E2 90.0722} C_DIS
LIN {X 8.113,Y 2.4988,Z 25,A -2.3331,B 0,C 0,E1 0.1598,E2 90.0721} C_DIS
LIN {X 8.3635,Y 1.4676,Z 25,A -2.3674,B 0,C 0,E1 0.1598,E2 90.0717} C_DIS
LIN {X 8.4844,Y 0.2674,Z 25,A -2.4139,B 0,C 0,E1 0.1598,E2 90.0716} C_DIS
LIN {X 8.4489,Y -0.8461,Z 25,A -2.4628,B 0,C 0,E1 0.1598,E2 90.0716} C_DIS
LIN {X 8.2749,Y -1.8891,Z 25,A -2.5137,B 0,C 0,E1 0.1598,E2 90.0716} C_DIS
LIN {X 8.0455,Y -2.7035,Z 25,A -2.557,B 0,C 0,E1 0.1598,E2 90.0718} C_DIS
LIN {X 7.7363,Y -3.4909,Z 25,A -2.6019,B 0,C 0,E1 0.1598,E2 90.0718} C_DIS
LIN {X 7.3503,Y -4.2437,Z 25,A -2.6482,B 0,C 0,E1 0.1598,E2 90.0718} C_DIS
LIN {X 6.8914,Y -4.9545,Z 25,A -2.6953,B 0,C 0,E1 0.1598,E2 90.0718} C_DIS
LIN {X 6.3641,Y -5.6161,Z 25,A -2.7429,B 0,C 0,E1 0.1598,E2 90.0717} C_DIS
LIN {X 5.7736,Y -6.2219,Z 25,A -2.7904,B 0,C 0,E1 0.1598,E2 90.0717} C_DIS
LIN {X 5.126,Y -6.7663,Z 25,A -2.8374,B 0,C 0,E1 0.1598,E2 90.0717} C_DIS
LIN {X 4.4273,Y -7.2433,Z 25,A -2.8833,B 0,C 0,E1 0.1598,E2 90.0717} C_DIS
LIN {X 3.6844,Y -7.6481,Z 25,A -2.9278,B 0,C 0,E1 0.1598,E2 90.0716} C_DIS
LIN {X 2.9049,Y -7.9768,Z 25,A -2.9704,B 0,C 0,E1 0.1598,E2 90.0716} C_DIS
LIN {X 2.0965,Y -8.2261,Z 25,A -3.0106,B 0,C 0,E1 0.1598,E2 90.0716} C_DIS
LIN {X 0.8412,Y -8.4495,Z 25,A -3.0661,B 0,C 0,E1 0.1598,E2 90.0715} C_DIS
LIN {X 0.8412,Y -8.4495,Z 25,A -3.0661,B 0,C 0,E1 0.1598,E2 90.0715} C_DIS
Enddeposition()
LIN {X 0.0007,Y -4.7572,Z 26,A -2.9252,B 0,C 0,E1 0.1598,E2 90.0603} C_DIS
Startdeposition()
$VEL.CP = VEL_PRINT
LIN {X 0.0007,Y -4.7572,Z 26,A -2.9309,B 0,C 0,E1 0.1598,E2 90.0661} C_DIS
LIN {X 0.9508,Y -4.654,Z 26,A -2.8966,B 0,C 0,E1 0.1598,E2 90.071} C_DIS
LIN {X 1.6848,Y -4.4405,Z 26,A -2.8611,B 0,C 0,E1 0.1598,E2 90.0717} C_DIS
LIN {X 2.3747,Y -4.1119,Z 26,A -2.8219,B 0,C 0,E1 0.1598,E2 90.0717} C_DIS
LIN {X 3.0046,Y -3.6789,Z 26,A -2.7803,B 0,C 0,E1 0.1598,E2 90.0717} C_DIS
LIN {X 3.5548,Y -3.1482,Z 26,A -2.7375,B 0,C 0,E1 0.1598,E2 90.0717} C_DIS
LIN {X 3.9091,Y -2.6973,Z 26,A -2.7053,B 0,C 0,E1 0.1598,E2 90.0718} C_DIS
LIN {X 4.2061,Y -2.2066,Z 26,A -2.6736,B 0,C 0,E1 0.1598,E2 90.0718} C_DIS
LIN {X 4.5046,Y -1.5029,Z 26,A -2.6325,B 0,C 0,E1 0.1598,E2 90.0718} C_DIS
LIN {X 4.688,Y -0.7611,Z 26,A -2.5942,B 0,C 0,E1 0.1598,E2 90.0718} C_DIS
LIN {X 4.75,Y 0.0008,Z 26,A -2.5595,B 0,C 0,E1 0.1598,E2 90.0718} C_DIS
LIN {X 4.6885,Y 0.7627,Z 26,A -2.5294,B 0,C 0,E1 0.1598,E2 90.0718} C_DIS
LIN {X 4.5047,Y 1.5046,Z 26,A -2.5047,B 0,C 0,E1 0.1598,E2 90.0719} C_DIS
LIN {X 4.2064,Y 2.2085,Z 26,A -2.4858,B 0,C 0,E1 0.1598,E2 90.0719} C_DIS
LIN {X 3.7984,Y 2.8553,Z 26,A -2.4734,B 0,C 0,E1 0.1598,E2 90.072} C_DIS
LIN {X 3.22,Y 3.4916,Z 26,A -2.4677,B 0,C 0,E1 0.1598,E2 90.072} C_DIS
LIN {X 2.6974,Y 3.9093,Z 26,A -2.4694,B 0,C 0,E1 0.1598,E2 90.0722} C_DIS
LIN {X 2.0355,Y 4.2918,Z 26,A -2.4776,B 0,C 0,E1 0.1598,E2 90.0722} C_DIS
LIN {X 1.321,Y 4.5638,Z 26,A -2.4924,B 0,C 0,E1 0.1598,E2 90.0722} C_DIS
LIN {X 0.5717,Y 4.7152,Z 26,A -2.5137,B 0,C 0,E1 0.1598,E2 90.0722} C_DIS
LIN {X -0.1921,Y 4.7448,Z 26,A -2.5406,B 0,C 0,E1 0.1598,E2 90.0722} C_DIS
LIN {X -0.951,Y 4.6536,Z 26,A -2.5724,B 0,C 0,E1 0.1598,E2 90.0722} C_DIS
LIN {X -1.6849,Y 4.4401,Z 26,A -2.6085,B 0,C 0,E1 0.1598,E2 90.0721} C_DIS
LIN {X -2.375,Y 4.1121,Z 26,A -2.6478,B 0,C 0,E1 0.1598,E2 90.072} C_DIS
LIN {X -3.0046,Y 3.6789,Z 26,A -2.6893,B 0,C 0,E1 0.1598,E2 90.0719} C_DIS
LIN {X -3.557,Y 3.1501,Z 26,A -2.7319,B 0,C 0,E1 0.1598,E2 90.0718} C_DIS
LIN {X -4.0168,Y 2.539,Z 26,A -2.7746,B 0,C 0,E1 0.1598,E2 90.0717} C_DIS
LIN {X -4.3712,Y 1.8614,Z 26,A -2.8162,B 0,C 0,E1 0.1598,E2 90.0716} C_DIS
LIN {X -4.6132,Y 1.1361,Z 26,A -2.8558,B 0,C 0,E1 0.1598,E2 90.0715} C_DIS
LIN {X -4.7356,Y 0.3814,Z 26,A -2.8921,B 0,C 0,E1 0.1598,E2 90.0715} C_DIS
LIN {X -4.7338,Y -0.3829,Z 26,A -2.9244,B 0,C 0,E1 0.1598,E2 90.0714} C_DIS
LIN {X -4.6537,Y -0.9509,Z 26,A -2.9456,B 0,C 0,E1 0.1598,E2 90.0714} C_DIS
LIN {X -4.4397,Y -1.6846,Z 26,A -2.9686,B 0,C 0,E1 0.1598,E2 90.0714} C_DIS
LIN {X -4.2054,Y -2.2079,Z 26,A -2.9822,B 0,C 0,E1 0.1598,E2 90.0714} C_DIS
LIN {X -3.7967,Y -2.8538,Z 26,A -2.9945,B 0,C 0,E1 0.1598,E2 90.0714} C_DIS
LIN {X -3.2893,Y -3.4256,Z 26,A -3.0001,B 0,C 0,E1 0.1598,E2 90.0714} C_DIS
LIN {X -2.6974,Y -3.9091,Z 26,A -2.9989,B 0,C 0,E1 0.1598,E2 90.0714} C_DIS
LIN {X -2.2066,Y -4.2061,Z 26,A -2.9935,B 0,C 0,E1 0.1598,E2 90.0715} C_DIS
LIN {X -1.503,Y -4.5045,Z 26,A -2.9803,B 0,C 0,E1 0.1598,E2 90.0715} C_DIS
LIN {X -0.9494,Y -4.654,Z 26,A -2.9664,B 0,C 0,E1 0.1598,E2 90.0716} C_DIS
LIN {X -0.1906,Y -4.7489,Z 26,A -2.9426,B 0,C 0,E1 0.1598,E2 90.0716} C_DIS
LIN {X -0.1906,Y -4.7489,Z 26,A -2.9426,B 0,C 0,E1 0.1598,E2 90.0716} C_DIS
Enddeposition()
LIN {X -0.0012,Y -5.6862,Z 26,A -2.9744,B 0,C 0,E1 0.1598,E2 90.0704} C_DIS
Startdeposition()
$VEL.CP = VEL_PRINT
LIN {X -0.7141,Y -5.6451,Z 26,A -2.9999,B 0,C 0,E1 0.1598,E2 90.0715} C_DIS
LIN {X -2.011,Y -5.3224,Z 26,A -3.0338,B 0,C 0,E1 0.1598,E2 90.0715} C_DIS
LIN {X -2.5774,Y -5.0672,Z 26,A -3.0438,B 0,C 0,E1 0.1598,E2 90.0715} C_DIS
LIN {X -3.2851,Y -4.6379,Z 26,A -3.0515,B 0,C 0,E1 0.1598,E2 90.0714} C_DIS
LIN {X -3.9243,Y -4.1122,Z 26,A -3.0527,B 0,C 0,E1 0.1598,E2 90.0714} C_DIS
LIN {X -4.4793,Y -3.4983,Z 26,A -3.047,B 0,C 0,E1 0.1598,E2 90.0714} C_DIS
LIN {X -4.9408,Y -2.8113,Z 26,A -3.0348,B 0,C 0,E1 0.1598,E2 90.0713} C_DIS
LIN {X -5.2961,Y -2.0638,Z 26,A -3.0162,B 0,C 0,E1 0.1598,E2 90.0713} C_DIS
LIN {X -5.5386,Y -1.2726,Z 26,A -2.9917,B 0,C 0,E1 0.1598,E2 90.0713} C_DIS
LIN {X -5.6647,Y -0.4549,Z 26,A -2.9617,B 0,C 0,E1 0.1598,E2 90.0713} C_DIS
LIN {X -5.6695,Y 0.3725,Z 26,A -2.927,B 0,C 0,E1 0.1598,E2 90.0713} C_DIS
LIN {X -5.5571,Y 1.1922,Z 26,A -2.8882,B 0,C 0,E1 0.1598,E2 90.0713} C_DIS
LIN {X -5.3262,Y 1.9869,Z 26,A -2.8462,B 0,C 0,E1 0.1598,E2 90.0715} C_DIS
LIN {X -4.9808,Y 2.7391,Z 26,A -2.8017,B 0,C 0,E1 0.1598,E2 90.0715} C_DIS
LIN {X -4.5313,Y 3.4341,Z 26,A -2.7558,B 0,C 0,E1 0.1598,E2 90.0717} C_DIS
LIN {X -3.9844,Y 4.0556,Z 26,A -2.7095,B 0,C 0,E1 0.1598,E2 90.0717} C_DIS
LIN {X -3.3527,Y 4.5902,Z 26,A -2.6636,B 0,C 0,E1 0.1598,E2 90.0719} C_DIS
LIN {X -2.6513,Y 5.0298,Z 26,A -2.6193,B 0,C 0,E1 0.1598,E2 90.0719} C_DIS
LIN {X -1.8929,Y 5.3616,Z 26,A -2.5773,B 0,C 0,E1 0.1598,E2 90.0721} C_DIS
LIN {X -1.0941,Y 5.5791,Z 26,A -2.5387,B 0,C 0,E1 0.1598,E2 90.0721} C_DIS
LIN {X -0.2724,Y 5.6798,Z 26,A -2.5041,B 0,C 0,E1 0.1598,E2 90.0722} C_DIS
LIN {X 0.4644,Y 5.6712,Z 26,A -2.4773,B 0,C 0,E1 0.1598,E2 90.0722} C_DIS
LIN {X 1.0639,Y 5.5831,Z 26,A -2.4589,B 0,C 0,E1 0.1598,E2 90.0722} C_DIS
LIN {X 1.8443,Y 5.3756,Z 26,A -2.4389,B 0,C 0,E1 0.1598,E2 90.0722} C_DIS
LIN {X 2.5882,Y 5.0616,Z 26,A -2.4248,B 0,C 0,E1 0.1598,E2 90.0722} C_DIS
LIN {X 3.28,Y 4.6446,Z 26,A -2.4169,B 0,C 0,E1 0.1598,E2 90.0722} C_DIS
LIN {X 3.9041,Y 4.1319,Z 26,A -2.4156,B 0,C 0,E1 0.1598,E2 90.0722} C_DIS
LIN {X 4.4497,Y 3.5364,Z 26,A -2.4207,B 0,C 0,E1 0.1598,E2 90.0722} C_DIS
LIN {X 4.9053,Y 2.8698,Z 26,A -2.4322,B 0,C 0,E1 0.1598,E2 90.0721} C_DIS
LIN {X 5.2623,Y 2.1456,Z 26,A -2.4497,B 0,C 0,E1 0.1598,E2 90.072} C_DIS
LIN {X 5.5969,Y 1.029,Z 26,A -2.4845,B 0,C 0,E1 0.1598,E2 90.0716} C_DIS
LIN {X 5.6874,Y 0.051,Z 26,A -2.5229,B 0,C 0,E1 0.1598,E2 90.0716} C_DIS
LIN {X 5.6569,Y -0.5695,Z 26,A -2.5507,B 0,C 0,E1 0.1598,E2 90.0719} C_DIS
LIN {X 5.4669,Y -1.5805,Z 26,A -2.6003,B 0,C 0,E1 0.1598,E2 90.0715} C_DIS
LIN {X 5.0952,Y -2.5318,Z 26,A -2.6545,B 0,C 0,E1 0.1598,E2 90.0715} C_DIS
LIN {X 4.2623,Y -3.7693,Z 26,A -2.7374,B 0,C 0,E1 0.1598,E2 90.0711} C_DIS
LIN {X 3.5917,Y -4.4067,Z 26,A -2.7897,B 0,C 0,E1 0.1598,E2 90.0716} C_DIS
LIN {X 2.9892,Y -4.837,Z 26,A -2.8302,B 0,C 0,E1 0.1598,E2 90.0717} C_DIS
LIN {X 2.3343,Y -5.1818,Z 26,A -2.8689,B 0,C 0,E1 0.1598,E2 90.0717} C_DIS
LIN {X 1.6418,Y -5.4432,Z 26,A -2.9055,B 0,C 0,E1 0.1598,E2 90.0717} C_DIS
LIN {X 0.9207,Y -5.6102,Z 26,A -2.9391,B 0,C 0,E1 0.1598,E2 90.0717} C_DIS
LIN {X -0.0012,Y -5.6862,Z 26,A -2.9761,B 0,C 0,E1 0.1598,E2 90.0717} C_DIS
Enddeposition()
LIN {X -0.0012,Y -5.6862,Z 26,A -2.9761,B 0,C 0,E1 0.1598,E2 90.0717} C_DIS
Startdeposition()
$VEL.CP = VEL_PRINT
LIN {X 0.5147,Y -6.5981,Z 26,A -2.9955,B 0,C 0,E1 0.1598,E2 90.071} C_DIS
LIN {X 1.2414,Y -6.5012,Z 26,A -2.9653,B 0,C 0,E1 0.1598,E2 90.0716} C_DIS
LIN {X 1.9529,Y -6.324,Z 26,A -2.9316,B 0,C 0,E1 0.1598,E2 90.0716} C_DIS
LIN {X 2.6404,Y -6.0692,Z 26,A -2.8956,B 0,C 0,E1 0.1598,E2 90.0716} C_DIS
LIN {X 3.2958,Y -5.7403,Z 26,A -2.8575,B 0,C 0,E1 0.1598,E2 90.0717} C_DIS
LIN {X 3.9109,Y -5.341,Z 26,A -2.818,B 0,C 0,E1 0.1598,E2 90.0717} C_DIS
LIN {X 4.4771,Y -4.8749,Z 26,A -2.7773,B 0,C 0,E1 0.1598,E2 90.0717} C_DIS
LIN {X 4.9884,Y -4.3493,Z 26,A -2.7362,B 0,C 0,E1 0.1598,E2 90.0717} C_DIS
LIN {X 5.4387,Y -3.7707,Z 26,A -2.695,B 0,C 0,E1 0.1598,E2 90.0718} C_DIS
LIN {X 5.8228,Y -3.1461,Z 26,A -2.6542,B 0,C 0,E1 0.1598,E2 90.0718} C_DIS
LIN {X 6.1342,Y -2.4823,Z 26,A -2.6145,B 0,C 0,E1 0.1598,E2 90.0718} C_DIS
LIN {X 6.3723,Y -1.7889,Z 26,A -2.5762,B 0,C 0,E1 0.1598,E2 90.0718} C_DIS
LIN {X 6.5313,Y -1.0731,Z 26,A -2.5399,B 0,C 0,E1 0.1598,E2 90.0719} C_DIS
LIN {X 6.6094,Y -0.344,Z 26,A -2.506,B 0,C 0,E1 0.1598,E2 90.0719} C_DIS
LIN {X 6.6066,Y 0.3891,Z 26,A -2.4749,B 0,C 0,E1 0.1598,E2 90.0719} C_DIS
LIN {X 6.5262,Y 1.1179,Z 26,A -2.4469,B 0,C 0,E1 0.1598,E2 90.072} C_DIS
LIN {X 6.3619,Y 1.8325,Z 26,A -2.4225,B 0,C 0,E1 0.1598,E2 90.072} C_DIS
LIN {X 6.1177,Y 2.5238,Z 26,A -2.4022,B 0,C 0,E1 0.1598,E2 90.072} C_DIS
LIN {X 5.8011,Y 3.1851,Z 26,A -2.3857,B 0,C 0,E1 0.1598,E2 90.0721} C_DIS
LIN {X 5.4156,Y 3.8089,Z 26,A -2.3735,B 0,C 0,E1 0.1598,E2 90.0721} C_DIS
LIN {X 4.9603,Y 4.3836,Z 26,A -2.3659,B 0,C 0,E1 0.1598,E2 90.0722} C_DIS
LIN {X 4.4452,Y 4.9057,Z 26,A -2.3627,B 0,C 0,E1 0.1598,E2 90.0722} C_DIS
LIN {X 3.8749,Y 5.3669,Z 26,A -2.3642,B 0,C 0,E1 0.1598,E2 90.0722} C_DIS
LIN {X 2.9648,Y 5.9228,Z 26,A -2.3742,B 0,C 0,E1 0.1598,E2 90.0722} C_DIS
LIN {X 2.0753,Y 6.2852,Z 26,A -2.3917,B 0,C 0,E1 0.1598,E2 90.0722} C_DIS
LIN {X 1.333,Y 6.4838,Z 26,A -2.4108,B 0,C 0,E1 0.1598,E2 90.0723} C_DIS
LIN {X 0.5726,Y 6.595,Z 26,A -2.4341,B 0,C 0,E1 0.1598,E2 90.0723} C_DIS
LIN {X -0.1954,Y 6.6149,Z 26,A -2.4616,B 0,C 0,E1 0.1598,E2 90.0723} C_DIS
LIN {X -0.9606,Y 6.5478,Z 26,A -2.4927,B 0,C 0,E1 0.1598,E2 90.0723} C_DIS
LIN {X -1.7137,Y 6.3952,Z 26,A -2.5269,B 0,C 0,E1 0.1598,E2 90.0722} C_DIS
LIN {X -2.4427,Y 6.1522,Z 26,A -2.5641,B 0,C 0,E1 0.1598,E2 90.0722} C_DIS
LIN {X -3.1394,Y 5.8278,Z 26,A -2.6035,B 0,C 0,E1 0.1598,E2 90.0721} C_DIS
LIN {X -3.7946,Y 5.4262,Z 26,A -2.6446,B 0,C 0,E1 0.1598,E2 90.072} C_DIS
LIN {X -4.397,Y 4.9491,Z 26,A -2.6869,B 0,C 0,E1 0.1598,E2 90.0719} C_DIS
LIN {X -4.9407,Y 4.4063,Z 26,A -2.7298,B 0,C 0,E1 0.1598,E2 90.0718} C_DIS
LIN {X -5.4188,Y 3.8048,Z 26,A -2.7728,B 0,C 0,E1 0.1598,E2 90.0717} C_DIS
LIN {X -5.8233,Y 3.1514,Z 26,A -2.8152,B 0,C 0,E1 0.1598,E2 90.0717} C_DIS
LIN {X -6.1482,Y 2.4551,Z 26,A -2.8566,B 0,C 0,E1 0.1598,E2 90.0715} C_DIS
LIN {X -6.3891,Y 1.7256,Z 26,A -2.8962,B 0,C 0,E1 0.1598,E2 90.0715} C_DIS
LIN {X -6.5459,Y 0.9735,Z 26,A -2.9337,B 0,C 0,E1 0.1598,E2 90.0714} C_DIS
LIN {X -6.6175,Y 0.2084,Z 26,A -2.9686,B 0,C 0,E1 0.1598,E2 90.0714} C_DIS
LIN {X -6.5947,Y -0.5597,Z 26,A -3.0002,B 0,C 0,E1 0.1598,E2 90.0713} C_DIS
LIN {X -6.4848,Y -1.32,Z 26,A -3.0283,B 0,C 0,E1 0.1598,E2 90.0713} C_DIS
LIN {X -6.289,Y -2.063,Z 26,A -3.0525,B 0,C 0,E1 0.1598,E2 90.0713} C_DIS
LIN {X -6.0073,Y -2.7778,Z 26,A -3.0723,B 0,C 0,E1 0.1598,E2 90.0713} C_DIS
LIN {X -5.644,Y -3.4547,Z 26,A -3.0876,B 0,C 0,E1 0.1598,E2 90.0713} C_DIS
LIN {X -5.2059,Y -4.0858,Z 26,A -3.0983,B 0,C 0,E1 0.1598,E2 90.0713} C_DIS
LIN {X -4.6971,Y -4.6614,Z 26,A -3.104,B 0,C 0,E1 0.1598,E2 90.0713} C_DIS
LIN {X -4.1268,Y -5.1763,Z 26,A -3.1049,B 0,C 0,E1 0.1598,E2 90.0713} C_DIS
LIN {X -3.5002,Y -5.621,Z 26,A -3.1007,B 0,C 0,E1 0.1598,E2 90.0713} C_DIS
LIN {X -2.825,Y -5.9879,Z 26,A -3.0915,B 0,C 0,E1 0.1598,E2 90.0713} C_DIS
LIN {X -2.1116,Y -6.2729,Z 26,A -3.0775,B 0,C 0,E1 0.1598,E2 90.0714} C_DIS
LIN {X -1.3702,Y -6.4744,Z 26,A -3.0589,B 0,C 0,E1 0.1598,E2 90.0714} C_DIS
LIN {X -0.6108,Y -6.5916,Z 26,A -3.036,B 0,C 0,E1 0.1598,E2 90.0715} C_DIS
LIN {X -0.6108,Y -6.5916,Z 26,A -3.036,B 0,C 0,E1 0.1598,E2 90.0715} C_DIS
Enddeposition()
LIN {X -0.069,Y -7.5567,Z 26,A -3.0561,B 0,C 0,E1 0.1598,E2 90.0703} C_DIS
Startdeposition()
$VEL.CP = VEL_PRINT
LIN {X -0.9858,Y -7.4885,Z 26,A -3.0879,B 0,C 0,E1 0.1598,E2 90.0714} C_DIS
LIN {X -2.0417,Y -7.277,Z 26,A -3.1177,B 0,C 0,E1 0.1598,E2 90.0714} C_DIS
LIN {X -3.0827,Y -6.8947,Z 26,A -3.1396,B 0,C 0,E1 0.1598,E2 90.0714} C_DIS
LIN {X -4.0614,Y -6.3731,Z 26,A -3.1533,B 0,C 0,E1 0.1598,E2 90.0712} C_DIS
LIN {X -4.9569,Y -5.6973,Z 26,A -3.1574,B 0,C 0,E1 0.1598,E2 90.0711} C_DIS
LIN {X -5.5492,Y -5.122,Z 26,A -3.1549,B 0,C 0,E1 0.1598,E2 90.0711} C_DIS
LIN {X -6.0755,Y -4.4856,Z 26,A -3.1473,B 0,C 0,E1 0.1598,E2 90.0711} C_DIS
LIN {X -6.5293,Y -3.7957,Z 26,A -3.1348,B 0,C 0,E1 0.1598,E2 90.0711} C_DIS
LIN {X -6.9056,Y -3.0607,Z 26,A -3.1175,B 0,C 0,E1 0.1598,E2 90.0711} C_DIS
LIN {X -7.197,Y -2.2881,Z 26,A -3.0955,B 0,C 0,E1 0.1598,E2 90.0711} C_DIS
LIN {X -7.4034,Y -1.4885,Z 26,A -3.0693,B 0,C 0,E1 0.1598,E2 90.0711} C_DIS
LIN {X -7.5493,Y -0.3667,Z 26,A -3.0271,B 0,C 0,E1 0.1598,E2 90.0709} C_DIS
LIN {X -7.5058,Y 0.8769,Z 26,A -2.9727,B 0,C 0,E1 0.1598,E2 90.0707} C_DIS
LIN {X -7.2793,Y 2.0129,Z 26,A -2.9166,B 0,C 0,E1 0.1598,E2 90.071} C_DIS
LIN {X -7.0063,Y 2.823,Z 26,A -2.8727,B 0,C 0,E1 0.1598,E2 90.0714} C_DIS
LIN {X -6.4699,Y 3.9047,Z 26,A -2.8071,B 0,C 0,E1 0.1598,E2 90.0713} C_DIS
LIN {X -5.8708,Y 4.7608,Z 26,A -2.7491,B 0,C 0,E1 0.1598,E2 90.0715} C_DIS
LIN {X -5.2101,Y 5.4731,Z 26,A -2.6947,B 0,C 0,E1 0.1598,E2 90.0717} C_DIS
LIN {X -4.4974,Y 6.0739,Z 26,A -2.6432,B 0,C 0,E1 0.1598,E2 90.0719} C_DIS
LIN {X -3.5395,Y 6.6772,Z 26,A -2.5824,B 0,C 0,E1 0.1598,E2 90.0719} C_DIS
LIN {X -2.4085,Y 7.1583,Z 26,A -2.5204,B 0,C 0,E1 0.1598,E2 90.0721} C_DIS
LIN {X -1.192,Y 7.4622,Z 26,A -2.4627,B 0,C 0,E1 0.1598,E2 90.0722} C_DIS
LIN {X -0.0814,Y 7.557,Z 26,A -2.4178,B 0,C 0,E1 0.1598,E2 90.0723} C_DIS
LIN {X 1.3597,Y 7.4352,Z 26,A -2.3697,B 0,C 0,E1 0.1598,E2 90.0723} C_DIS
LIN {X 2.5826,Y 7.0992,Z 26,A -2.3387,B 0,C 0,E1 0.1598,E2 90.0723} C_DIS
LIN {X 3.2925,Y 6.7991,Z 26,A -2.3253,B 0,C 0,E1 0.1598,E2 90.0724} C_DIS
LIN {X 4.1333,Y 6.3284,Z 26,A -2.3141,B 0,C 0,E1 0.1598,E2 90.0724} C_DIS
LIN {X 5.0786,Y 5.5905,Z 26,A -2.3103,B 0,C 0,E1 0.1598,E2 90.0721} C_DIS
LIN {X 5.6241,Y 5.0497,Z 26,A -2.3133,B 0,C 0,E1 0.1598,E2 90.0722} C_DIS
LIN {X 6.2876,Y 4.1929,Z 26,A -2.325,B 0,C 0,E1 0.1598,E2 90.072} C_DIS
LIN {X 6.8384,Y 3.2166,Z 26,A -2.3461,B 0,C 0,E1 0.1598,E2 90.0718} C_DIS
LIN {X 7.305,Y 1.9344,Z 26,A -2.383,B 0,C 0,E1 0.1598,E2 90.0714} C_DIS
LIN {X 7.5296,Y 0.6587,Z 26,A -2.4291,B 0,C 0,E1 0.1598,E2 90.0714} C_DIS
LIN {X 7.5347,Y -0.5836,Z 26,A -2.4817,B 0,C 0,E1 0.1598,E2 90.0714} C_DIS
LIN {X 7.3458,Y -1.7576,Z 26,A -2.5387,B 0,C 0,E1 0.1598,E2 90.0714} C_DIS
LIN {X 7.0929,Y -2.5981,Z 26,A -2.5842,B 0,C 0,E1 0.1598,E2 90.0717} C_DIS
LIN {X 6.7412,Y -3.4022,Z 26,A -2.6314,B 0,C 0,E1 0.1598,E2 90.0717} C_DIS
LIN {X 6.3022,Y -4.1621,Z 26,A -2.68,B 0,C 0,E1 0.1598,E2 90.0717} C_DIS
LIN {X 5.5318,Y -5.1482,Z 26,A -2.7501,B 0,C 0,E1 0.1598,E2 90.0714} C_DIS
LIN {X 4.5755,Y -6.0138,Z 26,A -2.822,B 0,C 0,E1 0.1598,E2 90.0714} C_DIS
LIN {X 3.4736,Y -6.7125,Z 26,A -2.8923,B 0,C 0,E1 0.1598,E2 90.0714} C_DIS
LIN {X 2.4841,Y -7.1378,Z 26,A -2.9469,B 0,C 0,E1 0.1598,E2 90.0716} C_DIS
LIN {X 1.4376,Y -7.4164,Z 26,A -2.9971,B 0,C 0,E1 0.1598,E2 90.0716} C_DIS
LIN {X 0.5038,Y -7.5401,Z 26,A -3.0366,B 0,C 0,E1 0.1598,E2 90.0716} C_DIS
LIN {X 0.5038,Y -7.5401,Z 26,A -3.0366,B 0,C 0,E1 0.1598,E2 90.0716} C_DIS
Enddeposition()
LIN {X -0.0932,Y -8.4898,Z 26,A -3.0979,B 0,C 0,E1 0.1598,E2 90.0703} C_DIS
Startdeposition()
$VEL.CP = VEL_PRINT
LIN {X 0.8417,Y -8.4494,Z 26,A -3.063,B 0,C 0,E1 0.1598,E2 90.0714} C_DIS
LIN {X 2.0897,Y -8.2278,Z 26,A -3.0079,B 0,C 0,E1 0.1598,E2 90.0715} C_DIS
LIN {X 2.8988,Y -7.979,Z 26,A -2.9677,B 0,C 0,E1 0.1598,E2 90.0715} C_DIS
LIN {X 3.679,Y -7.6506,Z 26,A -2.9251,B 0,C 0,E1 0.1598,E2 90.0716} C_DIS
LIN {X 4.4226,Y -7.246,Z 26,A -2.8806,B 0,C 0,E1 0.1598,E2 90.0716} C_DIS
LIN {X 5.1221,Y -6.7692,Z 26,A -2.8346,B 0,C 0,E1 0.1598,E2 90.0716} C_DIS
LIN {X 5.7703,Y -6.2248,Z 26,A -2.7876,B 0,C 0,E1 0.1598,E2 90.0717} C_DIS
LIN {X 6.3615,Y -5.6189,Z 26,A -2.74,B 0,C 0,E1 0.1598,E2 90.0717} C_DIS
LIN {X 6.8894,Y -4.9571,Z 26,A -2.6924,B 0,C 0,E1 0.1598,E2 90.0717} C_DIS
LIN {X 7.3489,Y -4.2461,Z 26,A -2.6452,B 0,C 0,E1 0.1598,E2 90.0717} C_DIS
LIN {X 7.7353,Y -3.493,Z 26,A -2.5989,B 0,C 0,E1 0.1598,E2 90.0718} C_DIS
LIN {X 8.0449,Y -2.7051,Z 26,A -2.554,B 0,C 0,E1 0.1598,E2 90.0718} C_DIS
LIN {X 8.2746,Y -1.8903,Z 26,A -2.5108,B 0,C 0,E1 0.1598,E2 90.0718} C_DIS
LIN {X 8.4489,Y -0.8466,Z 26,A -2.4596,B 0,C 0,E1 0.1598,E2 90.0716} C_DIS
LIN {X 8.4845,Y 0.2677,Z 26,A -2.4108,B 0,C 0,E1 0.1598,E2 90.0716} C_DIS
LIN {X 8.3647,Y 1.4601,Z 26,A -2.3643,B 0,C 0,E1 0.1598,E2 90.0716} C_DIS
LIN {X 8.1149,Y 2.4923,Z 26,A -2.3298,B 0,C 0,E1 0.1598,E2 90.0719} C_DIS
LIN {X 7.8252,Y 3.2911,Z 26,A -2.3067,B 0,C 0,E1 0.1598,E2 90.0721} C_DIS
LIN {X 7.457,Y 4.0568,Z 26,A -2.2877,B 0,C 0,E1 0.1598,E2 90.0721} C_DIS
LIN {X 7.0139,Y 4.7818,Z 26,A -2.2733,B 0,C 0,E1 0.1598,E2 90.0722} C_DIS
LIN {X 6.5004,Y 5.4588,Z 26,A -2.2635,B 0,C 0,E1 0.1598,E2 90.0722} C_DIS
LIN {X 5.9218,Y 6.081,Z 26,A -2.2584,B 0,C 0,E1 0.1598,E2 90.0723} C_DIS
LIN {X 5.2839,Y 6.6423,Z 26,A -2.2582,B 0,C 0,E1 0.1598,E2 90.0723} C_DIS
LIN {X 4.5931,Y 7.137,Z 26,A -2.2627,B 0,C 0,E1 0.1598,E2 90.0723} C_DIS
LIN {X 3.8566,Y 7.5608,Z 26,A -2.272,B 0,C 0,E1 0.1598,E2 90.0724} C_DIS
LIN {X 3.0813,Y 7.9086,Z 26,A -2.2859,B 0,C 0,E1 0.1598,E2 90.0724} C_DIS
LIN {X 2.2752,Y 8.1772,Z 26,A -2.3043,B 0,C 0,E1 0.1598,E2 90.0724} C_DIS
LIN {X 1.4463,Y 8.3642,Z 26,A -2.327,B 0,C 0,E1 0.1598,E2 90.0724} C_DIS
LIN {X 0.603,Y 8.4678,Z 26,A -2.3538,B 0,C 0,E1 0.1598,E2 90.0724} C_DIS
LIN {X -0.6547,Y 8.4656,Z 26,A -2.4003,B 0,C 0,E1 0.1598,E2 90.0724} C_DIS
LIN {X -1.6864,Y 8.3197,Z 26,A -2.4446,B 0,C 0,E1 0.1598,E2 90.0724} C_DIS
LIN {X -2.4941,Y 8.1136,Z 26,A -2.4831,B 0,C 0,E1 0.1598,E2 90.0722} C_DIS
LIN {X -3.5564,Y 7.7112,Z 26,A -2.5393,B 0,C 0,E1 0.1598,E2 90.0722} C_DIS
LIN {X -4.4937,Y 7.2008,Z 26,A -2.5954,B 0,C 0,E1 0.1598,E2 90.072} C_DIS
LIN {X -5.1942,Y 6.7127,Z 26,A -2.6418,B 0,C 0,E1 0.1598,E2 90.072} C_DIS
LIN {X -5.8422,Y 6.1567,Z 26,A -2.6891,B 0,C 0,E1 0.1598,E2 90.0718} C_DIS
LIN {X -6.4314,Y 5.5387,Z 26,A -2.7369,B 0,C 0,E1 0.1598,E2 90.0718} C_DIS
LIN {X -7.1608,Y 4.5627,Z 26,A -2.8047,B 0,C 0,E1 0.1598,E2 90.0714} C_DIS
LIN {X -7.7262,Y 3.5114,Z 26,A -2.8697,B 0,C 0,E1 0.1598,E2 90.0711} C_DIS
LIN {X -8.0418,Y 2.7134,Z 26,A -2.9152,B 0,C 0,E1 0.1598,E2 90.0713} C_DIS
LIN {X -8.3516,Y 1.539,Z 26,A -2.9758,B 0,C 0,E1 0.1598,E2 90.0709} C_DIS
LIN {X -8.4888,Y 0.1759,Z 26,A -3.0381,B 0,C 0,E1 0.1598,E2 90.0707} C_DIS
LIN {X -8.462,Y -0.7091,Z 26,A -3.0747,B 0,C 0,E1 0.1598,E2 90.0709} C_DIS
LIN {X -8.3232,Y -1.6778,Z 26,A -3.1105,B 0,C 0,E1 0.1598,E2 90.0709} C_DIS
LIN {X -8.0453,Y -2.7038,Z 26,A -3.1437,B 0,C 0,E1 0.1598,E2 90.0709} C_DIS
LIN {X -7.7343,Y -3.4954,Z 26,A -3.1658,B 0,C 0,E1 0.1598,E2 90.071} C_DIS
LIN {X -7.3455,Y -4.2518,Z 26,A -3.1836,B 0,C 0,E1 0.1598,E2 90.071} C_DIS
LIN {X -6.883,Y -4.9655,Z 26,A -3.1968,B 0,C 0,E1 0.1598,E2 90.071} C_DIS
LIN {X -6.1422,Y -5.8612,Z 26,A -3.2073,B 0,C 0,E1 0.1598,E2 90.071} C_DIS
LIN {X -5.2948,Y -6.6336,Z 26,A -3.209,B 0,C 0,E1 0.1598,E2 90.071} C_DIS
LIN {X -4.6188,Y -7.1202,Z 26,A -3.205,B 0,C 0,E1 0.1598,E2 90.0712} C_DIS
LIN {X -3.8985,Y -7.5383,Z 26,A -3.1963,B 0,C 0,E1 0.1598,E2 90.0712} C_DIS
LIN {X -3.1408,Y -7.884,Z 26,A -3.1832,B 0,C 0,E1 0.1598,E2 90.0712} C_DIS
LIN {X -2.3529,Y -8.1538,Z 26,A -3.1658,B 0,C 0,E1 0.1598,E2 90.0713} C_DIS
LIN {X -1.5424,Y -8.3453,Z 26,A -3.1442,B 0,C 0,E1 0.1598,E2 90.0713} C_DIS
LIN {X -0.7172,Y -8.4568,Z 26,A -3.1188,B 0,C 0,E1 0.1598,E2 90.0714} C_DIS
LIN {X -0.7172,Y -8.4568,Z 26,A -3.1188,B 0,C 0,E1 0.1598,E2 90.0714} C_DIS
Enddeposition()
LIN {X 0.0007,Y -4.757,Z 27,A -2.9204,B 0,C 0,E1 0.1598,E2 90.0604} C_DIS
Startdeposition()
$VEL.CP = VEL_PRINT
LIN {X 0.0007,Y -4.757,Z 27,A -2.9261,B 0,C 0,E1 0.1598,E2 90.0661} C_DIS
LIN {X -0.6752,Y -4.7017,Z 27,A -2.9534,B 0,C 0,E1 0.1598,E2 90.071} C_DIS
LIN {X -1.3375,Y -4.5574,Z 27,A -2.9723,B 0,C 0,E1 0.1598,E2 90.0716} C_DIS
LIN {X -2.06,Y -4.2792,Z 27,A -2.987,B 0,C 0,E1 0.1598,E2 90.0716} C_DIS
LIN {X -2.728,Y -3.8876,Z 27,A -2.9949,B 0,C 0,E1 0.1598,E2 90.0715} C_DIS
LIN {X -3.3232,Y -3.3926,Z 27,A -2.9957,B 0,C 0,E1 0.1598,E2 90.0715} C_DIS
LIN {X -3.8306,Y -2.8077,Z 27,A -2.9895,B 0,C 0,E1 0.1598,E2 90.0714} C_DIS
LIN {X -4.237,Y -2.1486,Z 27,A -2.9765,B 0,C 0,E1 0.1598,E2 90.0714} C_DIS
LIN {X -4.5299,Y -1.4318,Z 27,A -2.9569,B 0,C 0,E1 0.1598,E2 90.0714} C_DIS
LIN {X -4.7017,Y -0.6767,Z 27,A -2.9313,B 0,C 0,E1 0.1598,E2 90.0714} C_DIS
LIN {X -4.7506,Y 0.0962,Z 27,A -2.9004,B 0,C 0,E1 0.1598,E2 90.0714} C_DIS
LIN {X -4.6723,Y 0.8668,Z 27,A -2.8649,B 0,C 0,E1 0.1598,E2 90.0714} C_DIS
LIN {X -4.4674,Y 1.6137,Z 27,A -2.8259,B 0,C 0,E1 0.1598,E2 90.0715} C_DIS
LIN {X -4.1463,Y 2.3183,Z 27,A -2.7843,B 0,C 0,E1 0.1598,E2 90.0716} C_DIS
LIN {X -3.7155,Y 2.9619,Z 27,A -2.7413,B 0,C 0,E1 0.1598,E2 90.0717} C_DIS
LIN {X -3.1842,Y 3.5256,Z 27,A -2.6979,B 0,C 0,E1 0.1598,E2 90.0718} C_DIS
LIN {X -2.5682,Y 3.9948,Z 27,A -2.6554,B 0,C 0,E1 0.1598,E2 90.0719} C_DIS
LIN {X -1.885,Y 4.3593,Z 27,A -2.6149,B 0,C 0,E1 0.1598,E2 90.072} C_DIS
LIN {X -1.1516,Y 4.607,Z 27,A -2.5774,B 0,C 0,E1 0.1598,E2 90.0721} C_DIS
LIN {X -0.3879,Y 4.734,Z 27,A -2.5439,B 0,C 0,E1 0.1598,E2 90.0721} C_DIS
LIN {X 0.3865,Y 4.7336,Z 27,A -2.5153,B 0,C 0,E1 0.1598,E2 90.0722} C_DIS
LIN {X 1.1502,Y 4.6075,Z 27,A -2.4925,B 0,C 0,E1 0.1598,E2 90.0722} C_DIS
LIN {X 1.8838,Y 4.3598,Z 27,A -2.4759,B 0,C 0,E1 0.1598,E2 90.0722} C_DIS
LIN {X 2.5674,Y 3.9963,Z 27,A -2.4661,B 0,C 0,E1 0.1598,E2 90.0722} C_DIS
LIN {X 3.182,Y 3.5253,Z 27,A -2.4634,B 0,C 0,E1 0.1598,E2 90.0722} C_DIS
LIN {X 3.7126,Y 2.9615,Z 27,A -2.4677,B 0,C 0,E1 0.1598,E2 90.0721} C_DIS
LIN {X 4.1436,Y 2.3185,Z 27,A -2.4791,B 0,C 0,E1 0.1598,E2 90.0721} C_DIS
LIN {X 4.4665,Y 1.615,Z 27,A -2.497,B 0,C 0,E1 0.1598,E2 90.072} C_DIS
LIN {X 4.6684,Y 0.8675,Z 27,A -2.5213,B 0,C 0,E1 0.1598,E2 90.0719} C_DIS
LIN {X 4.7406,Y 0.2912,Z 27,A -2.5432,B 0,C 0,E1 0.1598,E2 90.0719} C_DIS
LIN {X 4.7336,Y -0.3863,Z 27,A -2.5722,B 0,C 0,E1 0.1598,E2 90.0719} C_DIS
LIN {X 4.6301,Y -1.0559,Z 27,A -2.6045,B 0,C 0,E1 0.1598,E2 90.0719} C_DIS
LIN {X 4.3967,Y -1.7941,Z 27,A -2.6444,B 0,C 0,E1 0.1598,E2 90.0718} C_DIS
LIN {X 4.0474,Y -2.4849,Z 27,A -2.6867,B 0,C 0,E1 0.1598,E2 90.0718} C_DIS
LIN {X 3.589,Y -3.1089,Z 27,A -2.7301,B 0,C 0,E1 0.1598,E2 90.0718} C_DIS
LIN {X 2.9997,Y -3.6827,Z 27,A -2.7762,B 0,C 0,E1 0.1598,E2 90.0718} C_DIS
LIN {X 2.4029,Y -4.0959,Z 27,A -2.8157,B 0,C 0,E1 0.1598,E2 90.0718} C_DIS
LIN {X 1.7059,Y -4.4331,Z 27,A -2.8557,B 0,C 0,E1 0.1598,E2 90.0718} C_DIS
LIN {X 0.963,Y -4.6518,Z 27,A -2.8923,B 0,C 0,E1 0.1598,E2 90.0717} C_DIS
LIN {X 0.1945,Y -4.7488,Z 27,A -2.9246,B 0,C 0,E1 0.1598,E2 90.0717} C_DIS
LIN {X 0.1945,Y -4.7488,Z 27,A -2.9246,B 0,C 0,E1 0.1598,E2 90.0717} C_DIS
Enddeposition()
LIN {X 0.0354,Y -5.6889,Z 27,A -2.9693,B 0,C 0,E1 0.1598,E2 90.0704} C_DIS
Startdeposition()
$VEL.CP = VEL_PRINT
LIN {X 1.0953,Y -5.5794,Z 27,A -2.9269,B 0,C 0,E1 0.1598,E2 90.0716} C_DIS
LIN {X 1.9166,Y -5.3513,Z 27,A -2.8871,B 0,C 0,E1 0.1598,E2 90.0716} C_DIS
LIN {X 2.6946,Y -5.0033,Z 27,A -2.8437,B 0,C 0,E1 0.1598,E2 90.0717} C_DIS
LIN {X 3.4128,Y -4.5446,Z 27,A -2.7978,B 0,C 0,E1 0.1598,E2 90.0717} C_DIS
LIN {X 4.0541,Y -3.9833,Z 27,A -2.7503,B 0,C 0,E1 0.1598,E2 90.0717} C_DIS
LIN {X 4.6042,Y -3.3325,Z 27,A -2.7024,B 0,C 0,E1 0.1598,E2 90.0717} C_DIS
LIN {X 5.0512,Y -2.6068,Z 27,A -2.655,B 0,C 0,E1 0.1598,E2 90.0717} C_DIS
LIN {X 5.3843,Y -1.8223,Z 27,A -2.6094,B 0,C 0,E1 0.1598,E2 90.0717} C_DIS
LIN {X 5.5973,Y -0.9968,Z 27,A -2.5664,B 0,C 0,E1 0.1598,E2 90.0717} C_DIS
LIN {X 5.6835,Y -0.1487,Z 27,A -2.5271,B 0,C 0,E1 0.1598,E2 90.0718} C_DIS
LIN {X 5.6423,Y 0.7028,Z 27,A -2.4924,B 0,C 0,E1 0.1598,E2 90.0718} C_DIS
LIN {X 5.4724,Y 1.5382,Z 27,A -2.4631,B 0,C 0,E1 0.1598,E2 90.0718} C_DIS
LIN {X 5.1805,Y 2.3391,Z 27,A -2.4399,B 0,C 0,E1 0.1598,E2 90.0719} C_DIS
LIN {X 4.7724,Y 3.0873,Z 27,A -2.4232,B 0,C 0,E1 0.1598,E2 90.072} C_DIS
LIN {X 4.2572,Y 3.7664,Z 27,A -2.4134,B 0,C 0,E1 0.1598,E2 90.072} C_DIS
LIN {X 3.6471,Y 4.3616,Z 27,A -2.4107,B 0,C 0,E1 0.1598,E2 90.0721} C_DIS
LIN {X 2.9535,Y 4.8573,Z 27,A -2.4153,B 0,C 0,E1 0.1598,E2 90.0721} C_DIS
LIN {X 2.1938,Y 5.2441,Z 27,A -2.4269,B 0,C 0,E1 0.1598,E2 90.0722} C_DIS
LIN {X 1.5926,Y 5.4631,Z 27,A -2.4399,B 0,C 0,E1 0.1598,E2 90.0722} C_DIS
LIN {X 0.3988,Y 5.6757,Z 27,A -2.4749,B 0,C 0,E1 0.1598,E2 90.0722} C_DIS
LIN {X -0.7559,Y 5.64,Z 27,A -2.519,B 0,C 0,E1 0.1598,E2 90.0722} C_DIS
LIN {X -2.266,Y 5.2188,Z 27,A -2.5925,B 0,C 0,E1 0.1598,E2 90.072} C_DIS
LIN {X -3.512,Y 4.4761,Z 27,A -2.6696,B 0,C 0,E1 0.1598,E2 90.0717} C_DIS
LIN {X -3.9765,Y 4.0621,Z 27,A -2.7043,B 0,C 0,E1 0.1598,E2 90.0718} C_DIS
LIN {X -4.5246,Y 3.44,Z 27,A -2.7508,B 0,C 0,E1 0.1598,E2 90.0718} C_DIS
LIN {X -4.9779,Y 2.7458,Z 27,A -2.7967,B 0,C 0,E1 0.1598,E2 90.0716} C_DIS
LIN {X -5.3986,Y 1.7986,Z 27,A -2.8519,B 0,C 0,E1 0.1598,E2 90.0712} C_DIS
LIN {X -5.6718,Y 0.457,Z 27,A -2.9182,B 0,C 0,E1 0.1598,E2 90.0707} C_DIS
LIN {X -5.6611,Y -0.5279,Z 27,A -2.9599,B 0,C 0,E1 0.1598,E2 90.0711} C_DIS
LIN {X -5.5339,Y -1.3057,Z 27,A -2.9883,B 0,C 0,E1 0.1598,E2 90.0713} C_DIS
LIN {X -5.2982,Y -2.0577,Z 27,A -3.0114,B 0,C 0,E1 0.1598,E2 90.0713} C_DIS
LIN {X -4.9623,Y -2.7702,Z 27,A -3.0292,B 0,C 0,E1 0.1598,E2 90.0713} C_DIS
LIN {X -4.5305,Y -3.4291,Z 27,A -3.0413,B 0,C 0,E1 0.1598,E2 90.0713} C_DIS
LIN {X -4.0131,Y -4.0229,Z 27,A -3.0474,B 0,C 0,E1 0.1598,E2 90.0713} C_DIS
LIN {X -3.4191,Y -4.5405,Z 27,A -3.0476,B 0,C 0,E1 0.1598,E2 90.0713} C_DIS
LIN {X -2.5874,Y -5.0682,Z 27,A -3.0394,B 0,C 0,E1 0.1598,E2 90.0713} C_DIS
LIN {X -1.4495,Y -5.5018,Z 27,A -3.0161,B 0,C 0,E1 0.1598,E2 90.0714} C_DIS
LIN {X -0.7129,Y -5.6421,Z 27,A -2.9951,B 0,C 0,E1 0.1598,E2 90.0716} C_DIS
LIN {X 0.0354,Y -5.6889,Z 27,A -2.9697,B 0,C 0,E1 0.1598,E2 90.0716} C_DIS
Enddeposition()
LIN {X 0.0354,Y -5.6889,Z 27,A -2.9697,B 0,C 0,E1 0.1598,E2 90.0716} C_DIS
Startdeposition()
$VEL.CP = VEL_PRINT
LIN {X -0.5077,Y -6.5976,Z 27,A -3.0277,B 0,C 0,E1 0.1598,E2 90.071} C_DIS
LIN {X -1.2502,Y -6.5001,Z 27,A -3.0514,B 0,C 0,E1 0.1598,E2 90.0715} C_DIS
LIN {X -1.9772,Y -6.3195,Z 27,A -3.0704,B 0,C 0,E1 0.1598,E2 90.0715} C_DIS
LIN {X -2.6775,Y -6.0542,Z 27,A -3.0848,B 0,C 0,E1 0.1598,E2 90.0715} C_DIS
LIN {X -3.3443,Y -5.7128,Z 27,A -3.0948,B 0,C 0,E1 0.1598,E2 90.0714} C_DIS
LIN {X -3.9682,Y -5.2983,Z 27,A -3.1001,B 0,C 0,E1 0.1598,E2 90.0714} C_DIS
LIN {X -4.5415,Y -4.8163,Z 27,A -3.1007,B 0,C 0,E1 0.1598,E2 90.0714} C_DIS
LIN {X -5.0555,Y -4.2716,Z 27,A -3.0965,B 0,C 0,E1 0.1598,E2 90.0713} C_DIS
LIN {X -5.5067,Y -3.6738,Z 27,A -3.0877,B 0,C 0,E1 0.1598,E2 90.0713} C_DIS
LIN {X -5.8865,Y -3.0282,Z 27,A -3.0743,B 0,C 0,E1 0.1598,E2 90.0713} C_DIS
LIN {X -6.1899,Y -2.3434,Z 27,A -3.0565,B 0,C 0,E1 0.1598,E2 90.0713} C_DIS
LIN {X -6.4151,Y -1.6291,Z 27,A -3.0346,B 0,C 0,E1 0.1598,E2 90.0713} C_DIS
Enddeposition()
END
